// TIA Portal project "Lift_2026" (V15.1)

(* hardware
DEVICE "S71500/ET200MP station_1"  S7-1500 station
   slot 0: "Rail_0"  Rack  6ES7 590-1***0-0AA0
   slot 1: "PLC_1"  CPU 1513-1 PN  6ES7 513-1AL02-0AB0  V2.6
      slot 3: "CPU display_1"  6ES7591-1AA00-0AA0
DEVICE "HMI_1"  KTP900 Basic PN
   slot 0: "HMI_1"  KTP900 Basic PN  6AV2 123-2JB03-0AX0  15.1.0.0
   slot 1: "HMI_RT_1"  KTP900 Basic PN  6AV2 123-2JB03-0AX0  15.1.0.0
   slot 5: "HMI_1.IE_CP_1"  PROFINET Interface  15.0.1.0
      slot 1: "PROFINET Interface_1"  PROFINET Interface
         slot 1: "Port_1"  Port
*)

// ===== PLC "PLC_1"  CPU 1513-1 PN =====

VAR_GLOBAL   // PLC tag table "Default tag table"
   "Clock_Byte" AT %MB0 : Byte;
   "Clock_10Hz" AT %M0.0 : Bool;
   "Clock_5Hz" AT %M0.1 : Bool;
   "Clock_2.5Hz" AT %M0.2 : Bool;
   "Clock_2Hz" AT %M0.3 : Bool;
   "Clock_1.25Hz" AT %M0.4 : Bool;
   "Clock_1Hz" AT %M0.5 : Bool;
   "Clock_0.625Hz" AT %M0.6 : Bool;
   "Clock_0.5Hz" AT %M0.7 : Bool;
END_VAR

DATA_BLOCK "Alarme"   // DB1
{ S7_Optimized_Access := 'TRUE' }
VERSION : 0.1
   VAR
      alarme_gather : Word;
      alarme_vect : Array[0..15] of Bool;
   END_VAR
BEGIN
END_DATA_BLOCK

DATA_BLOCK "Avarii"   // DB2
{ S7_Optimized_Access := 'TRUE' }
VERSION : 0.1
   VAR
      esd : Bool;
      btn_esd : Bool;
      reset_esd : Bool;
      avarie_generala : Bool;
      reset_avarie_generala : Bool;
      avarie_usa : Bool;
      avarie_lumina : Bool;
      avarie_motor : Bool;
      avarie_greutate : Bool;
   END_VAR
BEGIN
END_DATA_BLOCK

DATA_BLOCK "Usa_Lift_DB"   // DB3
{ S7_Optimized_Access := 'TRUE' }
VERSION : 0.1
   VAR
      btn_urgenta : Bool;
      deschide_usa : Bool;
      inchide_usa : Bool;
      usa_deschisa : Bool;
      usa_inchisa : Bool;
   END_VAR
BEGIN
END_DATA_BLOCK

DATA_BLOCK "Bec_DB"   // DB4
{ S7_Optimized_Access := 'TRUE' }
VERSION : 0.1
   VAR
      permisiune_pornire : Bool;
      led_aprins : Bool;
   END_VAR
BEGIN
END_DATA_BLOCK

DATA_BLOCK "Motor_DB"   // DB5
{ S7_Optimized_Access := 'TRUE' }
VERSION : 0.1
   VAR
      pornire_stea : Bool;
      pornire_triunghi : Bool;
      directie_sus : Bool;
      directie_jos : Bool;
      permisiune_plecare : Bool;
   END_VAR
BEGIN
END_DATA_BLOCK

DATA_BLOCK "Simulare_DB"   // DB6
{ S7_Optimized_Access := 'TRUE' }
VERSION : 0.1
   VAR
      directie : USInt;
      etaj_curent : Int := 1;
      etaj_dorit : Int;
      etaj_chemat : Int;
      lift_in_miscare : Bool;
      btn_chemare_1 : Bool;
      btn_chemare_2 : Bool;
      btn_chemare_3 : Bool;
      btn_lift_1 : Bool;
      btn_lift_2 : Bool;
      btn_lift_3 : Bool;
      btn_add_pers : Bool;
      btn_sub_pers : Bool;
      time_elapsed_1 : Time;
      time_elapsed_2 : Time;
      time_elapsed_3 : Time;
      time_elapsed_4 : Time;
      time_elapsed_secunde_1 : Time;
      time_elapsed_secunde_2 : Time;
      time_elapsed_secunde_3 : Time;
      time_elapsed_secunde_4 : Time;
      "10s_cerut" : Bool;
      "10s_dorit" : Bool;
   END_VAR
BEGIN
END_DATA_BLOCK

DATA_BLOCK "Senzor_greutate_DB"   // DB7
{ S7_Optimized_Access := 'TRUE' }
VERSION : 0.1
   VAR
      permisiune_plecare : Bool := true;
      greutate_maxima : Real := 300.0;
      greutate_curenta : Real;
      greutate_depasita : Bool;
   END_VAR
BEGIN
END_DATA_BLOCK

DATA_BLOCK "Bec_DB_1"   // DB10
{ S7_Optimized_Access := 'TRUE' }
VERSION : 0.1
// stored: InstanceOfName Bec
"Bec"
BEGIN
END_DATA_BLOCK

DATA_BLOCK "Usa_Lift_DB_1"   // DB11
{ S7_Optimized_Access := 'TRUE' }
VERSION : 0.1
// stored: InstanceOfName Usa
"Usa"
BEGIN
END_DATA_BLOCK

DATA_BLOCK "Usa_Et_1_DB"   // DB12
{ S7_Optimized_Access := 'TRUE' }
VERSION : 0.1
   VAR
      deschide_usa : Bool;
      inchide_usa : Bool;
      usa_deschisa : Bool;
      usa_inchisa : Bool;
      btn_urgenta : Bool;
   END_VAR
BEGIN
END_DATA_BLOCK

DATA_BLOCK "USa_Et_2_DB"   // DB13
{ S7_Optimized_Access := 'TRUE' }
VERSION : 0.1
   VAR
      btn_urgenta : Bool;
      deschide_usa : Bool;
      inchide_usa : Bool;
      usa_deschisa : Bool;
      usa_inchisa : Bool;
   END_VAR
BEGIN
END_DATA_BLOCK

DATA_BLOCK "Usa_Et_3_DB"   // DB14
{ S7_Optimized_Access := 'TRUE' }
VERSION : 0.1
   VAR
      btn_urgenta : Bool;
      deschide_usa : Bool;
      inchide_usa : Bool;
      usa_deschisa : Bool;
      usa_inchisa : Bool;
   END_VAR
BEGIN
END_DATA_BLOCK

DATA_BLOCK "Usa_Et_1_DB_1"   // DB15
{ S7_Optimized_Access := 'TRUE' }
VERSION : 0.1
// stored: InstanceOfName Usa
"Usa"
BEGIN
END_DATA_BLOCK

DATA_BLOCK "Usa_Et_2_DB_1"   // DB16
{ S7_Optimized_Access := 'TRUE' }
VERSION : 0.1
// stored: InstanceOfName Usa
"Usa"
BEGIN
END_DATA_BLOCK

DATA_BLOCK "Usa_Et_3_DB_1"   // DB17
{ S7_Optimized_Access := 'TRUE' }
VERSION : 0.1
// stored: InstanceOfName Usa
"Usa"
BEGIN
END_DATA_BLOCK

DATA_BLOCK "Senzor_greutate_DB_1"   // DB18
{ S7_Optimized_Access := 'TRUE' }
VERSION : 0.1
// stored: InstanceOfName Senzor_greutate
"Senzor_greutate"
BEGIN
END_DATA_BLOCK

DATA_BLOCK "Motor_DB_1"   // DB19
{ S7_Optimized_Access := 'TRUE' }
VERSION : 0.1
// stored: InstanceOfName Motor
"Motor"
BEGIN
END_DATA_BLOCK

DATA_BLOCK "Simulare_DB_1"   // DB20
{ S7_Optimized_Access := 'TRUE' }
VERSION : 0.1
// stored: InstanceOfName Simulare
"Simulare"
BEGIN
END_DATA_BLOCK

// folder: System blocks/Program resources

DATA_BLOCK "timer_reset_esd"   // DB8
{ S7_Optimized_Access := 'TRUE' }
AUTHOR : Simatic
FAMILY : IEC
NAME : IEC_TMR
VERSION : 1.0
// stored: InstanceOfName IEC_TIMER
"IEC_TIMER"
BEGIN
END_DATA_BLOCK

DATA_BLOCK "timer_reset_avarie_generala"   // DB9
{ S7_Optimized_Access := 'TRUE' }
AUTHOR : Simatic
FAMILY : IEC
NAME : IEC_TMR
VERSION : 1.0
// stored: InstanceOfName IEC_TIMER
"IEC_TIMER"
BEGIN
END_DATA_BLOCK

// folder: (top level)

FUNCTION_BLOCK "Usa"   // FB1, LAD
{ S7_Optimized_Access := 'TRUE' }
VERSION : 0.1
   VAR_OUTPUT
      usa_deschisa : Bool;
      usa_inchisa : Bool;
   END_VAR
   VAR_IN_OUT
      deschide_usa : Bool;
      inchide_usa : Bool;
   END_VAR
   VAR
      timer_usa_inchisa : TON_TIME;
      timer_usa_deschisa : TON_TIME;
   END_VAR
BEGIN

REGION Network 1: deschide usa
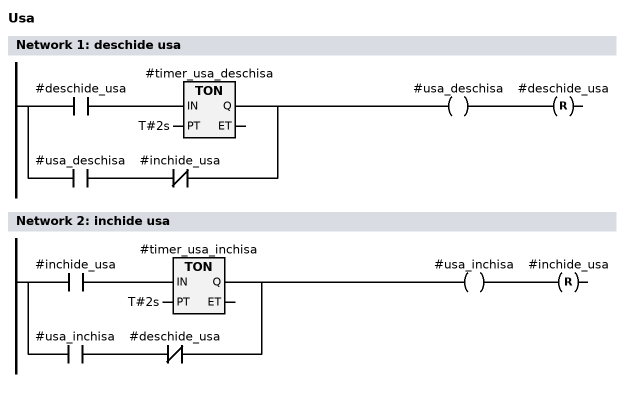
   #timer_usa_deschisa(IN := #deschide_usa, PT := T#2s);   // TON
   #usa_deschisa := #timer_usa_deschisa.Q OR (#usa_deschisa AND NOT #inchide_usa);
   IF #usa_deschisa THEN #deschide_usa := FALSE; END_IF;
END_REGION

REGION Network 2: inchide usa
   #timer_usa_inchisa(IN := #inchide_usa, PT := T#2s);   // TON
   #usa_inchisa := #timer_usa_inchisa.Q OR (#usa_inchisa AND NOT #deschide_usa);
   IF #usa_inchisa THEN #inchide_usa := FALSE; END_IF;
END_REGION
END_FUNCTION_BLOCK

FUNCTION_BLOCK "Bec"   // FB2, LAD
{ S7_Optimized_Access := 'TRUE' }
VERSION : 0.1
   VAR_INPUT
      permisiune_pornire : Bool;
   END_VAR
   VAR_OUTPUT
      bec_aprins : Bool;
   END_VAR
BEGIN

REGION Network 1
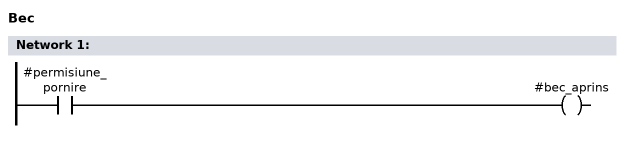
   RUNG wire#powerrail
      Contact( #permisiune_pornire )
      Coil( #bec_aprins )
   END_RUNG
   // the same network as SCL:
   #bec_aprins := #permisiune_pornire;
END_REGION
END_FUNCTION_BLOCK

FUNCTION_BLOCK "Motor"   // FB3, LAD
{ S7_Optimized_Access := 'TRUE' }
VERSION : 0.1
   VAR_INPUT
      directie : USInt;
   END_VAR
   VAR_OUTPUT
      pornire_stea : Bool;
      pornire_triunghi : Bool;
      directie_sus : Bool;
      directie_jos : Bool;
   END_VAR
   VAR_IN_OUT
      permisiune_plecare : Bool;
   END_VAR
   VAR
      timer_stea : TON_TIME;
   END_VAR
BEGIN

REGION Network 1: Selecteaza directia
   // simulata cu valori algebrice, insa in mod normal ar fi un contact pentru directie, depinzand cum se conecteaza, selecteaza directia, insa pentru simplitate am optat la asta
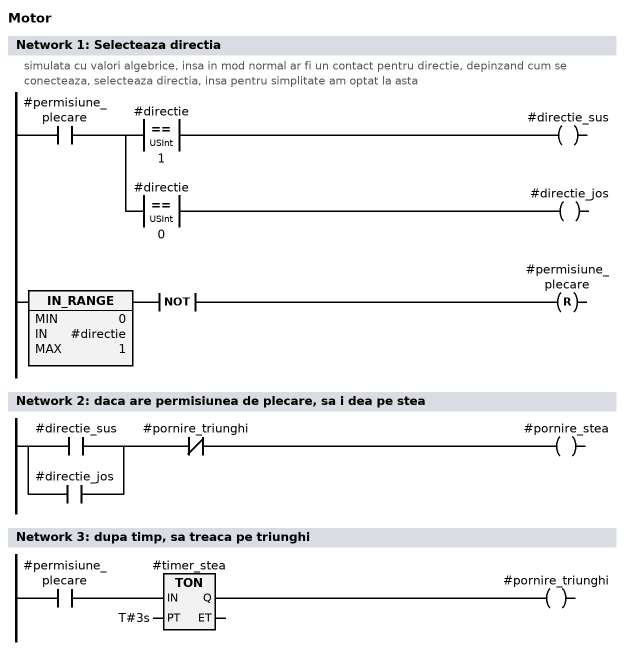
   RUNG wire#powerrail
      Contact( #permisiune_plecare )
      wire#w1
      { S7_Templates := "SrcType := USInt" } EQ_Contact(in1 := #directie, in2 := 1)
      Coil( #directie_sus )
   END_RUNG
   RUNG wire#w1
      { S7_Templates := "SrcType := USInt" } EQ_Contact(in1 := #directie, in2 := 0)
      Coil( #directie_jos )
   END_RUNG
   RUNG wire#powerrail
      { S7_Templates := "SrcType := USInt" } InRange(min := 0, in := #directie, max := 1)
      Not()
      R_Coil( #permisiune_plecare )
   END_RUNG
   // the same network as SCL:
   #directie_sus := #permisiune_plecare AND (#directie = 1);
   #directie_jos := #permisiune_plecare AND (#directie = 0);
   IF NOT ((0 <= #directie) AND (#directie <= 1)) THEN #permisiune_plecare := FALSE; END_IF;
END_REGION

REGION Network 2: daca are permisiunea de plecare, sa i dea pe stea
   RUNG wire#powerrail
      Contact( #directie_sus )
      wire#w1
      I_Contact( #pornire_triunghi )
      Coil( #pornire_stea )
   END_RUNG
   RUNG wire#powerrail
      Contact( #directie_jos )
   END_RUNG wire#w1
   // the same network as SCL:
   #pornire_stea := (#directie_sus OR #directie_jos) AND NOT #pornire_triunghi;
END_REGION

REGION Network 3: dupa timp, sa treaca pe triunghi
   #timer_stea(IN := #permisiune_plecare, PT := T#3s);   // TON
   #pornire_triunghi := #timer_stea.Q;
END_REGION
END_FUNCTION_BLOCK

FUNCTION_BLOCK "Simulare"   // FB4, LAD
{ S7_Optimized_Access := 'TRUE' }
VERSION : 0.1
   VAR_INPUT
      motor_pornit : Bool;
      greutate_maxima : Real;
      greutate_depasita : Bool;
      esd : Bool;
      avarie_generala : Bool;
      este_deschis_1 : Bool;
      este_deschis_2 : Bool;
      este_deschis_3 : Bool;
   END_VAR
   VAR_OUTPUT
      directie : USInt;
      lift_in_miscare : Bool;
      time_elapsed_dorit_1 : Time;
      time_elapsed_dorit_2 : Time;
      time_elapsed_cerut_1 : Time;
      time_elapsed_cerut_2 : Time;
      "10s_dorit" : Bool;
      "10s_cerut" : Bool;
   END_VAR
   VAR_IN_OUT
      btn_urgenta_usa_1 : Bool;
      btn_urgenta_usa_2 : Bool;
      btn_urgenta_usa_3 : Bool;
      btn_urgenta_usa_lift : Bool;
      btn_add_pers : Bool;
      btn_sub_pers : Bool;
      usa_lift_inchisa : Bool;
      usa_lift_deschisa : Bool;
      usa_deschisa_et_1 : Bool;
      usa_deschisa_et_2 : Bool;
      usa_deschisa_et_3 : Bool;
      usa_inchisa_et_1 : Bool;
      usa_inchisa_et_2 : Bool;
      usa_inchisa_et_3 : Bool;
      plecare_motor : Bool;
      plecare_greutate : Bool;
      plecare_lumina : Bool;
      btn_chemare_1 : Bool;
      btn_chemare_2 : Bool;
      btn_chemare_3 : Bool;
      btn_lift_1 : Bool;
      btn_lift_2 : Bool;
      btn_lift_3 : Bool;
      etaj_curent : Int;
      etaj_dorit : Int;
      etaj_chemat : Int;
      greutate_curenta : Real;
   END_VAR
   VAR
      ajuns_chemare : Bool;
      plecare : Bool;
      terminat_proces : Bool;
      timer_5s_chemat : TON_TIME;
      timer_10s_chemat : TON_TIME;
      timer_5s_plecat : TON_TIME;
      timer_10s_plecat : TON_TIME;
      timer_resetare_terminare : TON_TIME;
      add : Bool;
      sub : Bool;
      diferenta_chemat : Int;
      diferenta_plecat : Int;
      re_add : Bool;
      re_sub : Bool;
      trm_5s_plecat : Bool;
      trm_10s_plecat : Bool;
      trm_plecat : Bool;
      trm_5s_chemat : Bool;
      trm_10s_chemat : Bool;
      trm_chemat : Bool;
   END_VAR
   VAR_TEMP   // added for the SCL form of the ladder/FBD networks
      _w1 : Bool;
      _w2 : Bool;
      _w3 : Bool;
   END_VAR
BEGIN

REGION Network 1: seteaza ca liftul e in miscare
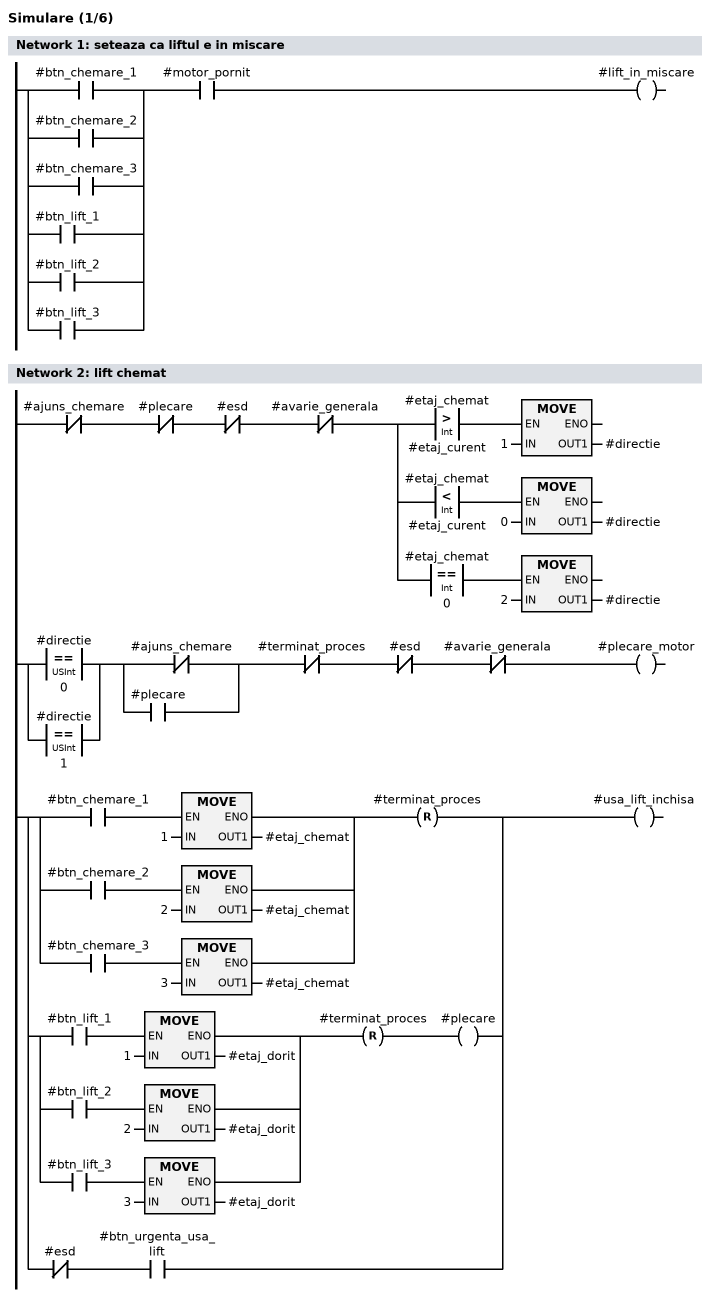
   RUNG wire#powerrail
      Contact( #btn_chemare_1 )
      wire#w1
      Contact( #motor_pornit )
      Coil( #lift_in_miscare )
   END_RUNG
   RUNG wire#powerrail
      Contact( #btn_chemare_2 )
   END_RUNG wire#w1
   RUNG wire#powerrail
      Contact( #btn_chemare_3 )
   END_RUNG wire#w1
   RUNG wire#powerrail
      Contact( #btn_lift_1 )
   END_RUNG wire#w1
   RUNG wire#powerrail
      Contact( #btn_lift_2 )
   END_RUNG wire#w1
   RUNG wire#powerrail
      Contact( #btn_lift_3 )
   END_RUNG wire#w1
   // the same network as SCL:
   #lift_in_miscare := (#btn_chemare_1 OR #btn_chemare_2 OR #btn_chemare_3 OR #btn_lift_1 OR #btn_lift_2 OR #btn_lift_3) AND #motor_pornit;
END_REGION

REGION Network 2: lift chemat
   RUNG wire#powerrail
      I_Contact( #ajuns_chemare )
      I_Contact( #plecare )
      I_Contact( #esd )
      I_Contact( #avarie_generala )
      wire#w1
      { S7_Templates := "SrcType := Int" } GT_Contact(in1 := #etaj_chemat, in2 := #etaj_curent)
      Move(in := 1, out1 => #directie)
   END_RUNG
   RUNG wire#w1
      { S7_Templates := "SrcType := Int" } LT_Contact(in1 := #etaj_chemat, in2 := #etaj_curent)
      Move(in := 0, out1 => #directie)
   END_RUNG
   RUNG wire#w1
      { S7_Templates := "SrcType := Int" } EQ_Contact(in1 := #etaj_chemat, in2 := 0)
      Move(in := 2, out1 => #directie)
   END_RUNG
   RUNG wire#powerrail
      { S7_Templates := "SrcType := USInt" } EQ_Contact(in1 := #directie, in2 := 0)
      wire#w2
      I_Contact( #ajuns_chemare )
      wire#w3
      I_Contact( #terminat_proces )
      I_Contact( #esd )
      I_Contact( #avarie_generala )
      Coil( #plecare_motor )
   END_RUNG
   RUNG wire#powerrail
      { S7_Templates := "SrcType := USInt" } EQ_Contact(in1 := #directie, in2 := 1)
   END_RUNG wire#w2
   RUNG wire#w2
      Contact( #plecare )
   END_RUNG wire#w3
   RUNG wire#powerrail
      Contact( #btn_chemare_1 )
      Move(in := 1, out1 => #etaj_chemat)
      wire#w4
      R_Coil( #terminat_proces )
      wire#w5
      Coil( #usa_lift_inchisa )
   END_RUNG
   RUNG wire#powerrail
      Contact( #btn_chemare_2 )
      Move(in := 2, out1 => #etaj_chemat)
   END_RUNG wire#w4
   RUNG wire#powerrail
      Contact( #btn_chemare_3 )
      Move(in := 3, out1 => #etaj_chemat)
   END_RUNG wire#w4
   RUNG wire#powerrail
      Contact( #btn_lift_1 )
      Move(in := 1, out1 => #etaj_dorit)
      wire#w6
      R_Coil( #terminat_proces )
      Coil( #plecare )
   END_RUNG wire#w5
   RUNG wire#powerrail
      Contact( #btn_lift_2 )
      Move(in := 2, out1 => #etaj_dorit)
   END_RUNG wire#w6
   RUNG wire#powerrail
      Contact( #btn_lift_3 )
      Move(in := 3, out1 => #etaj_dorit)
   END_RUNG wire#w6
   RUNG wire#powerrail
      I_Contact( #esd )
      Contact( #btn_urgenta_usa_lift )
   END_RUNG wire#w5
   // the same network as SCL:
   #_w1 := NOT #ajuns_chemare AND NOT #plecare AND NOT #esd AND NOT #avarie_generala;
   IF #_w1 AND (#etaj_chemat > #etaj_curent) THEN #directie := 1; END_IF;
   IF #_w1 AND (#etaj_chemat < #etaj_curent) THEN #directie := 0; END_IF;
   IF #_w1 AND (#etaj_chemat = 0) THEN #directie := 2; END_IF;
   #plecare_motor := ((#directie = 0) OR (#directie = 1)) AND (NOT #ajuns_chemare OR #plecare) AND NOT #terminat_proces AND NOT #esd AND NOT #avarie_generala;
   IF #btn_chemare_1 THEN #etaj_chemat := 1; END_IF;
   IF #btn_chemare_2 THEN #etaj_chemat := 2; END_IF;
   IF #btn_chemare_3 THEN #etaj_chemat := 3; END_IF;
   #_w2 := #btn_chemare_1 OR #btn_chemare_2 OR #btn_chemare_3;
   IF #_w2 THEN #terminat_proces := FALSE; END_IF;
   IF #btn_lift_1 THEN #etaj_dorit := 1; END_IF;
   IF #btn_lift_2 THEN #etaj_dorit := 2; END_IF;
   IF #btn_lift_3 THEN #etaj_dorit := 3; END_IF;
   #_w3 := #btn_lift_1 OR #btn_lift_2 OR #btn_lift_3;
   IF #_w3 THEN #terminat_proces := FALSE; END_IF;
   #plecare := #_w3;
   #usa_lift_inchisa := #_w2 OR #_w3 OR (NOT #esd AND #btn_urgenta_usa_lift);
END_REGION

REGION Network 3: daca simte persoana, aprinde lumina (pentru simplitate :) ), si calculeaza si diferenta, cuz why not
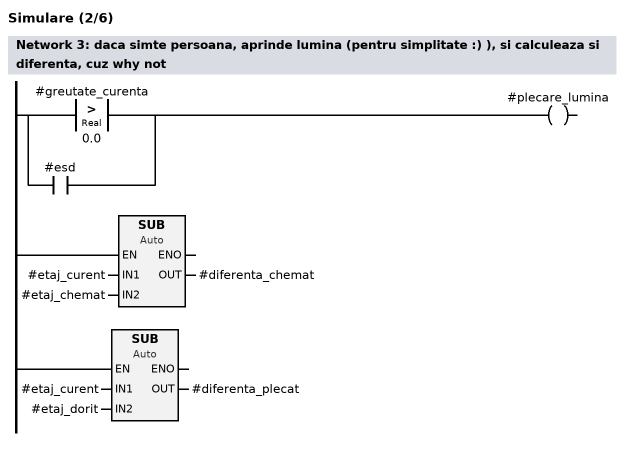
   RUNG wire#powerrail
      { S7_Templates := "SrcType := Real" } GT_Contact(in1 := #greutate_curenta, in2 := 0.0)
      wire#w1
      Coil( #plecare_lumina )
   END_RUNG
   RUNG wire#powerrail
      Contact( #esd )
   END_RUNG wire#w1
   RUNG wire#powerrail
      Sub(in1 := #etaj_curent, in2 := #etaj_chemat, out => #diferenta_chemat)
   END_RUNG
   RUNG wire#powerrail
      Sub(in1 := #etaj_curent, in2 := #etaj_dorit, out => #diferenta_plecat)
   END_RUNG
   // the same network as SCL:
   #plecare_lumina := (#greutate_curenta > 0.0) OR #esd;
   #diferenta_chemat := #etaj_curent - #etaj_chemat;
   #diferenta_plecat := #etaj_curent - #etaj_dorit;
END_REGION

REGION Network 4: daca a pornit motorul, depinzand de diferenta, pune ton ul
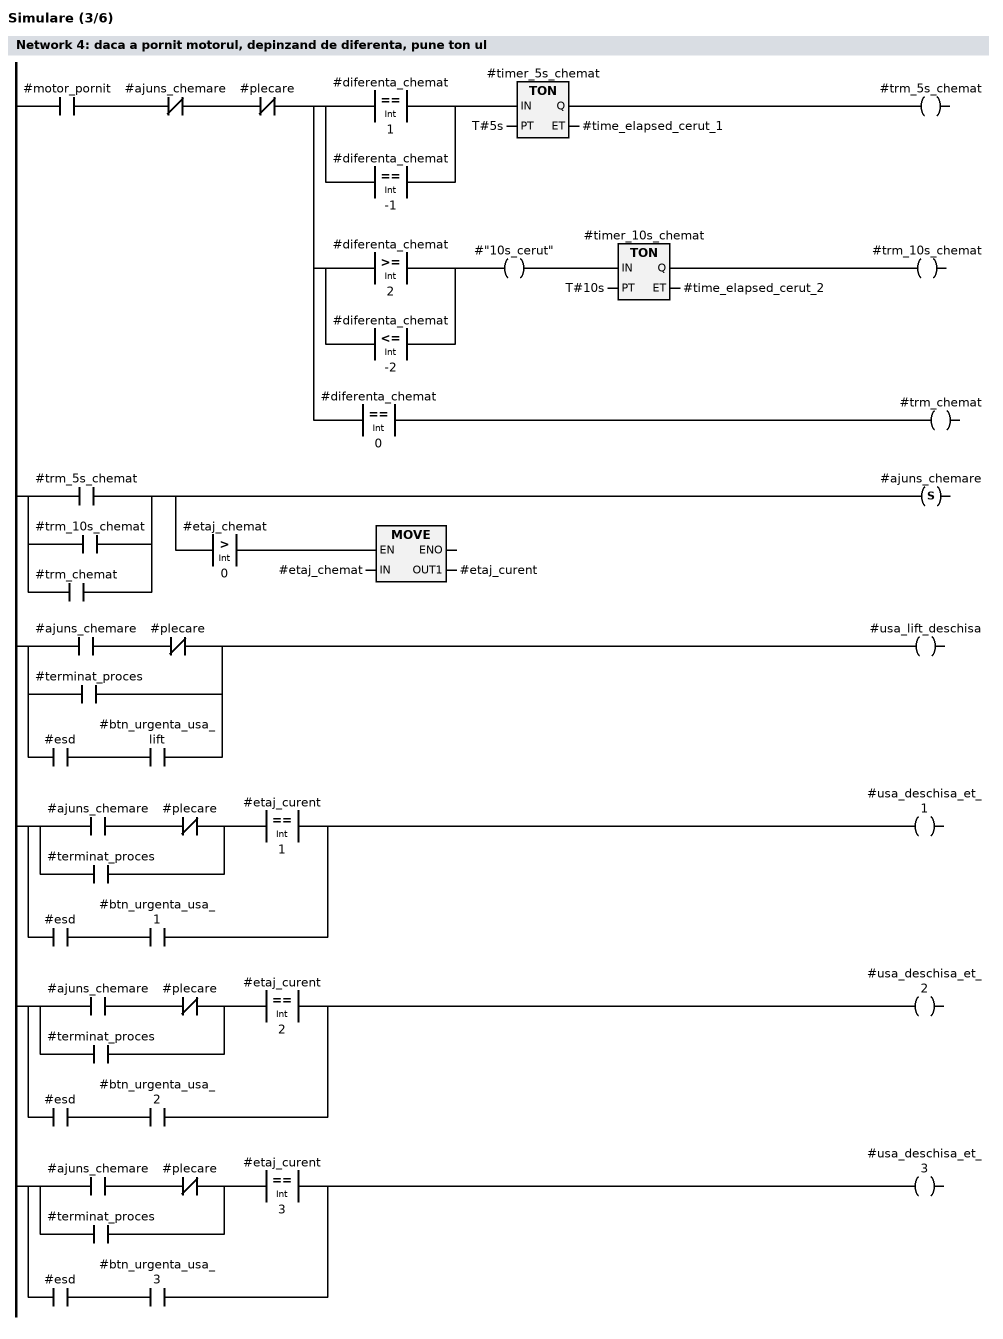
   #_w1 := #motor_pornit AND NOT #ajuns_chemare AND NOT #plecare;
   #timer_5s_chemat(IN := #_w1 AND ((#diferenta_chemat = 1) OR (#diferenta_chemat = (-1))),   // TON
                    PT := T#5s,
                    ET => #time_elapsed_cerut_1);
   #trm_5s_chemat := #timer_5s_chemat.Q;
   #"10s_cerut" := #_w1 AND ((#diferenta_chemat >= 2) OR (#diferenta_chemat <= (-2)));
   #timer_10s_chemat(IN := #"10s_cerut", PT := T#10s, ET => #time_elapsed_cerut_2);   // TON
   #trm_10s_chemat := #timer_10s_chemat.Q;
   #trm_chemat := #_w1 AND (#diferenta_chemat = 0);
   #_w2 := #trm_5s_chemat OR #trm_10s_chemat OR #trm_chemat;
   IF #_w2 THEN #ajuns_chemare := TRUE; END_IF;
   IF #_w2 AND (#etaj_chemat > 0) THEN #etaj_curent := #etaj_chemat; END_IF;
   #usa_lift_deschisa := (#ajuns_chemare AND NOT #plecare) OR #terminat_proces OR (#esd AND #btn_urgenta_usa_lift);
   #usa_deschisa_et_1 := (((#ajuns_chemare AND NOT #plecare) OR #terminat_proces) AND (#etaj_curent = 1)) OR (#esd AND #btn_urgenta_usa_1);
   #usa_deschisa_et_2 := (((#ajuns_chemare AND NOT #plecare) OR #terminat_proces) AND (#etaj_curent = 2)) OR (#esd AND #btn_urgenta_usa_2);
   #usa_deschisa_et_3 := (((#ajuns_chemare AND NOT #plecare) OR #terminat_proces) AND (#etaj_curent = 3)) OR (#esd AND #btn_urgenta_usa_3);
END_REGION

REGION Network 5: daca ii da buton din lift, sa plece la fel
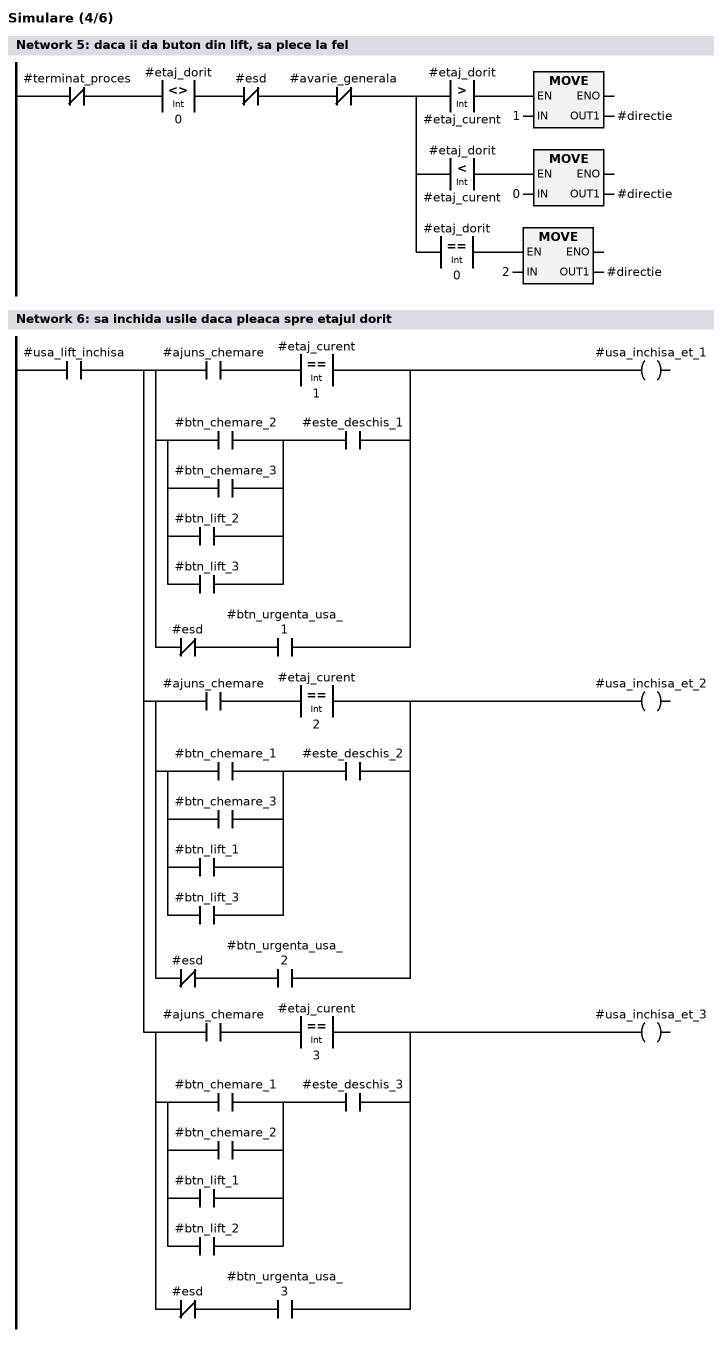
   RUNG wire#powerrail
      I_Contact( #terminat_proces )
      { S7_Templates := "SrcType := Int" } NE_Contact(in1 := #etaj_dorit, in2 := 0)
      I_Contact( #esd )
      I_Contact( #avarie_generala )
      wire#w1
      { S7_Templates := "SrcType := Int" } GT_Contact(in1 := #etaj_dorit, in2 := #etaj_curent)
      Move(in := 1, out1 => #directie)
   END_RUNG
   RUNG wire#w1
      { S7_Templates := "SrcType := Int" } LT_Contact(in1 := #etaj_dorit, in2 := #etaj_curent)
      Move(in := 0, out1 => #directie)
   END_RUNG
   RUNG wire#w1
      { S7_Templates := "SrcType := Int" } EQ_Contact(in1 := #etaj_dorit, in2 := 0)
      Move(in := 2, out1 => #directie)
   END_RUNG
   // the same network as SCL:
   #_w1 := NOT #terminat_proces AND (#etaj_dorit <> 0) AND NOT #esd AND NOT #avarie_generala;
   IF #_w1 AND (#etaj_dorit > #etaj_curent) THEN #directie := 1; END_IF;
   IF #_w1 AND (#etaj_dorit < #etaj_curent) THEN #directie := 0; END_IF;
   IF #_w1 AND (#etaj_dorit = 0) THEN #directie := 2; END_IF;
END_REGION

REGION Network 6: sa inchida usile daca pleaca spre etajul dorit
   RUNG wire#powerrail
      Contact( #usa_lift_inchisa )
      wire#w1
      Contact( #ajuns_chemare )
      { S7_Templates := "SrcType := Int" } EQ_Contact(in1 := #etaj_curent, in2 := 1)
      wire#w2
      Coil( #usa_inchisa_et_1 )
   END_RUNG
   RUNG wire#w1
      Contact( #btn_chemare_2 )
      wire#w3
      Contact( #este_deschis_1 )
   END_RUNG wire#w2
   RUNG wire#w1
      Contact( #btn_chemare_3 )
   END_RUNG wire#w3
   RUNG wire#w1
      Contact( #btn_lift_2 )
   END_RUNG wire#w3
   RUNG wire#w1
      Contact( #btn_lift_3 )
   END_RUNG wire#w3
   RUNG wire#w1
      I_Contact( #esd )
      Contact( #btn_urgenta_usa_1 )
   END_RUNG wire#w2
   RUNG wire#w1
      Contact( #ajuns_chemare )
      { S7_Templates := "SrcType := Int" } EQ_Contact(in1 := #etaj_curent, in2 := 2)
      wire#w4
      Coil( #usa_inchisa_et_2 )
   END_RUNG
   RUNG wire#w1
      Contact( #btn_chemare_1 )
      wire#w5
      Contact( #este_deschis_2 )
   END_RUNG wire#w4
   RUNG wire#w1
      Contact( #btn_chemare_3 )
   END_RUNG wire#w5
   RUNG wire#w1
      Contact( #btn_lift_1 )
   END_RUNG wire#w5
   RUNG wire#w1
      Contact( #btn_lift_3 )
   END_RUNG wire#w5
   RUNG wire#w1
      I_Contact( #esd )
      Contact( #btn_urgenta_usa_2 )
   END_RUNG wire#w4
   RUNG wire#w1
      Contact( #ajuns_chemare )
      { S7_Templates := "SrcType := Int" } EQ_Contact(in1 := #etaj_curent, in2 := 3)
      wire#w6
      Coil( #usa_inchisa_et_3 )
   END_RUNG
   RUNG wire#w1
      Contact( #btn_chemare_1 )
      wire#w7
      Contact( #este_deschis_3 )
   END_RUNG wire#w6
   RUNG wire#w1
      Contact( #btn_chemare_2 )
   END_RUNG wire#w7
   RUNG wire#w1
      Contact( #btn_lift_1 )
   END_RUNG wire#w7
   RUNG wire#w1
      Contact( #btn_lift_2 )
   END_RUNG wire#w7
   RUNG wire#w1
      I_Contact( #esd )
      Contact( #btn_urgenta_usa_3 )
   END_RUNG wire#w6
   // the same network as SCL:
   #usa_inchisa_et_1 := #usa_lift_inchisa AND ((#ajuns_chemare AND (#etaj_curent = 1)) OR ((#btn_chemare_2 OR #btn_chemare_3 OR #btn_lift_2 OR #btn_lift_3) AND #este_deschis_1) OR (NOT #esd AND #btn_urgenta_usa_1));
   #usa_inchisa_et_2 := #usa_lift_inchisa AND ((#ajuns_chemare AND (#etaj_curent = 2)) OR ((#btn_chemare_1 OR #btn_chemare_3 OR #btn_lift_1 OR #btn_lift_3) AND #este_deschis_2) OR (NOT #esd AND #btn_urgenta_usa_2));
   #usa_inchisa_et_3 := #usa_lift_inchisa AND ((#ajuns_chemare AND (#etaj_curent = 3)) OR ((#btn_chemare_1 OR #btn_chemare_2 OR #btn_lift_1 OR #btn_lift_2) AND #este_deschis_3) OR (NOT #esd AND #btn_urgenta_usa_3));
END_REGION

REGION Network 7: daca a pornit motorul, sa mearga la etajul dorit
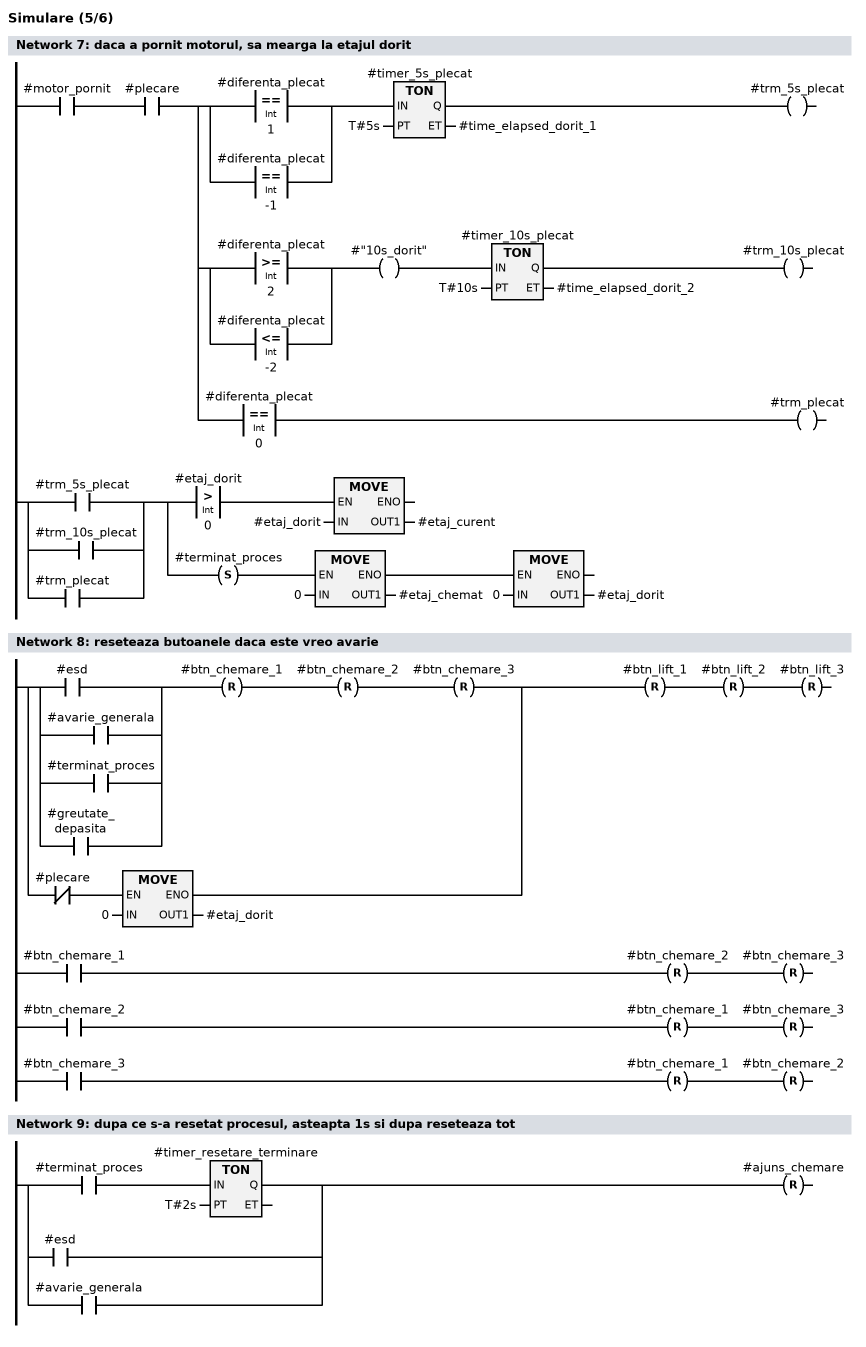
   #_w1 := #motor_pornit AND #plecare;
   #timer_5s_plecat(IN := #_w1 AND ((#diferenta_plecat = 1) OR (#diferenta_plecat = (-1))),   // TON
                    PT := T#5s,
                    ET => #time_elapsed_dorit_1);
   #trm_5s_plecat := #timer_5s_plecat.Q;
   #"10s_dorit" := #_w1 AND ((#diferenta_plecat >= 2) OR (#diferenta_plecat <= (-2)));
   #timer_10s_plecat(IN := #"10s_dorit", PT := T#10s, ET => #time_elapsed_dorit_2);   // TON
   #trm_10s_plecat := #timer_10s_plecat.Q;
   #trm_plecat := #_w1 AND (#diferenta_plecat = 0);
   #_w2 := #trm_5s_plecat OR #trm_10s_plecat OR #trm_plecat;
   IF #_w2 AND (#etaj_dorit > 0) THEN #etaj_curent := #etaj_dorit; END_IF;
   IF #_w2 THEN
       #terminat_proces := TRUE;
       #etaj_chemat := 0;
       #etaj_dorit := 0;
   END_IF;
END_REGION

REGION Network 8: reseteaza butoanele daca este vreo avarie
   RUNG wire#powerrail
      Contact( #esd )
      wire#w1
      R_Coil( #btn_chemare_1 )
      R_Coil( #btn_chemare_2 )
      R_Coil( #btn_chemare_3 )
      wire#w2
      R_Coil( #btn_lift_1 )
      R_Coil( #btn_lift_2 )
      R_Coil( #btn_lift_3 )
   END_RUNG
   RUNG wire#powerrail
      Contact( #avarie_generala )
   END_RUNG wire#w1
   RUNG wire#powerrail
      Contact( #terminat_proces )
   END_RUNG wire#w1
   RUNG wire#powerrail
      Contact( #greutate_depasita )
   END_RUNG wire#w1
   RUNG wire#powerrail
      I_Contact( #plecare )
      Move(in := 0, out1 => #etaj_dorit)
   END_RUNG wire#w2
   RUNG wire#powerrail
      Contact( #btn_chemare_1 )
      R_Coil( #btn_chemare_2 )
      R_Coil( #btn_chemare_3 )
   END_RUNG
   RUNG wire#powerrail
      Contact( #btn_chemare_2 )
      R_Coil( #btn_chemare_1 )
      R_Coil( #btn_chemare_3 )
   END_RUNG
   RUNG wire#powerrail
      Contact( #btn_chemare_3 )
      R_Coil( #btn_chemare_1 )
      R_Coil( #btn_chemare_2 )
   END_RUNG
   // the same network as SCL:
   #_w1 := #esd OR #avarie_generala OR #terminat_proces OR #greutate_depasita;
   IF #_w1 THEN
       #btn_chemare_1 := FALSE;
       #btn_chemare_2 := FALSE;
       #btn_chemare_3 := FALSE;
   END_IF;
   IF NOT #plecare THEN #etaj_dorit := 0; END_IF;
   IF #_w1 OR NOT #plecare THEN
       #btn_lift_1 := FALSE;
       #btn_lift_2 := FALSE;
       #btn_lift_3 := FALSE;
   END_IF;
   IF #btn_chemare_1 THEN
       #btn_chemare_2 := FALSE;
       #btn_chemare_3 := FALSE;
   END_IF;
   IF #btn_chemare_2 THEN
       #btn_chemare_1 := FALSE;
       #btn_chemare_3 := FALSE;
   END_IF;
   IF #btn_chemare_3 THEN
       #btn_chemare_1 := FALSE;
       #btn_chemare_2 := FALSE;
   END_IF;
END_REGION

REGION Network 9: dupa ce s-a resetat procesul, asteapta 1s si dupa reseteaza tot
   #timer_resetare_terminare(IN := #terminat_proces, PT := T#2s);   // TON
   IF #timer_resetare_terminare.Q OR #esd OR #avarie_generala THEN #ajuns_chemare := FALSE; END_IF;
END_REGION

REGION Network 10: butoane pt a adauga/scoate persoane din lift
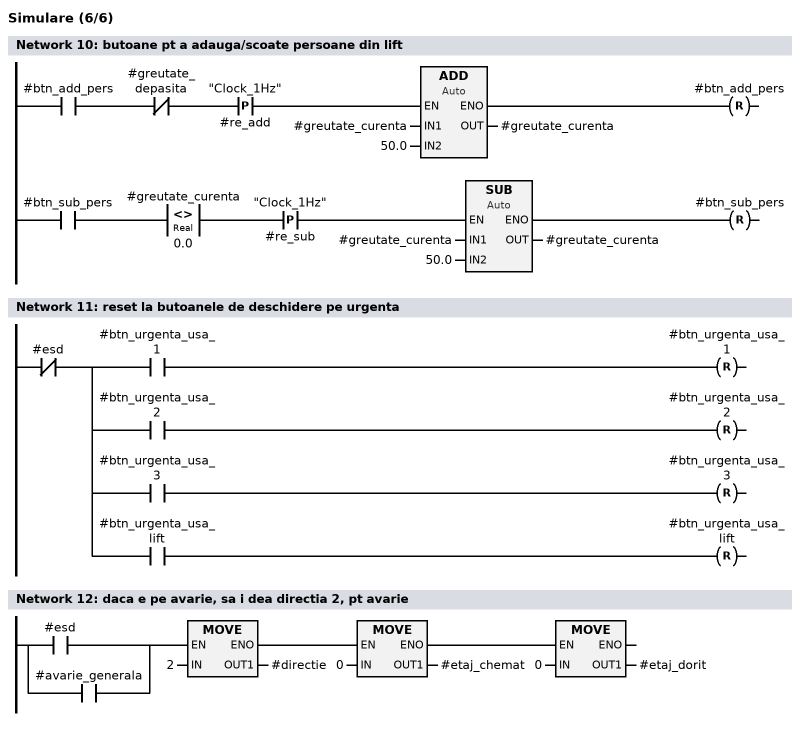
   RUNG wire#powerrail
      Contact( #btn_add_pers )
      I_Contact( #greutate_depasita )
      P_Contact(operand := "Clock_1Hz", bit := #re_add)
      Add(in1 := #greutate_curenta, in2 := 50.0, out => #greutate_curenta)
      R_Coil( #btn_add_pers )
   END_RUNG
   RUNG wire#powerrail
      Contact( #btn_sub_pers )
      { S7_Templates := "SrcType := Real" } NE_Contact(in1 := #greutate_curenta, in2 := 0.0)
      P_Contact(operand := "Clock_1Hz", bit := #re_sub)
      Sub(in1 := #greutate_curenta, in2 := 50.0, out => #greutate_curenta)
      R_Coil( #btn_sub_pers )
   END_RUNG
   // the same network as SCL:
   #_w1 := #btn_add_pers AND NOT #greutate_depasita AND "Clock_1Hz" AND NOT #re_add;   // rising edge of "Clock_1Hz"
   #re_add := "Clock_1Hz";
   IF #_w1 THEN
       #greutate_curenta := #greutate_curenta + 50.0;
       #btn_add_pers := FALSE;
   END_IF;
   #_w2 := #btn_sub_pers AND (#greutate_curenta <> 0.0) AND "Clock_1Hz" AND NOT #re_sub;   // rising edge of "Clock_1Hz"
   #re_sub := "Clock_1Hz";
   IF #_w2 THEN
       #greutate_curenta := #greutate_curenta - 50.0;
       #btn_sub_pers := FALSE;
   END_IF;
END_REGION

REGION Network 11: reset la butoanele de deschidere pe urgenta
   RUNG wire#powerrail
      I_Contact( #esd )
      wire#w1
      Contact( #btn_urgenta_usa_1 )
      R_Coil( #btn_urgenta_usa_1 )
   END_RUNG
   RUNG wire#w1
      Contact( #btn_urgenta_usa_2 )
      R_Coil( #btn_urgenta_usa_2 )
   END_RUNG
   RUNG wire#w1
      Contact( #btn_urgenta_usa_3 )
      R_Coil( #btn_urgenta_usa_3 )
   END_RUNG
   RUNG wire#w1
      Contact( #btn_urgenta_usa_lift )
      R_Coil( #btn_urgenta_usa_lift )
   END_RUNG
   // the same network as SCL:
   IF NOT #esd AND #btn_urgenta_usa_1 THEN #btn_urgenta_usa_1 := FALSE; END_IF;
   IF NOT #esd AND #btn_urgenta_usa_2 THEN #btn_urgenta_usa_2 := FALSE; END_IF;
   IF NOT #esd AND #btn_urgenta_usa_3 THEN #btn_urgenta_usa_3 := FALSE; END_IF;
   IF NOT #esd AND #btn_urgenta_usa_lift THEN #btn_urgenta_usa_lift := FALSE; END_IF;
END_REGION

REGION Network 12: daca e pe avarie, sa i dea directia 2, pt avarie
   RUNG wire#powerrail
      Contact( #esd )
      wire#w1
      Move(in := 2, out1 => #directie)
      Move(in := 0, out1 => #etaj_chemat)
      Move(in := 0, out1 => #etaj_dorit)
   END_RUNG
   RUNG wire#powerrail
      Contact( #avarie_generala )
   END_RUNG wire#w1
   // the same network as SCL:
   IF #esd OR #avarie_generala THEN
       #directie := 2;
       #etaj_chemat := 0;
       #etaj_dorit := 0;
   END_IF;
END_REGION
END_FUNCTION_BLOCK

FUNCTION_BLOCK "Senzor_greutate"   // FB5, LAD
{ S7_Optimized_Access := 'TRUE' }
VERSION : 0.1
   VAR_INPUT
      permisiune_plecare : Bool;
      greutate_maxima : Real;
   END_VAR
   VAR_OUTPUT
      greutate_depasita : Bool;
   END_VAR
   VAR_IN_OUT
      greutate_curenta : Real;
   END_VAR
   VAR
      pornit : Bool;
   END_VAR
BEGIN

REGION Network 1: daca are permisiune de plecare,
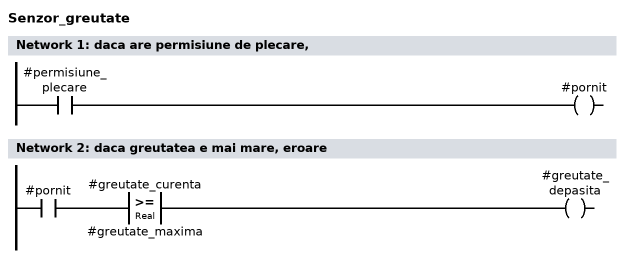
   RUNG wire#powerrail
      Contact( #permisiune_plecare )
      Coil( #pornit )
   END_RUNG
   // the same network as SCL:
   #pornit := #permisiune_plecare;
END_REGION

REGION Network 2: daca greutatea e mai mare, eroare
   RUNG wire#powerrail
      Contact( #pornit )
      { S7_Templates := "SrcType := Real" } GE_Contact(in1 := #greutate_curenta, in2 := #greutate_maxima)
      Coil( #greutate_depasita )
   END_RUNG
   // the same network as SCL:
   #greutate_depasita := #pornit AND (#greutate_curenta >= #greutate_maxima);
END_REGION
END_FUNCTION_BLOCK

ORGANIZATION_BLOCK "Main"   // OB1, LAD, ProgramCycle
TITLE = "Main Program Sweep (Cycle)"
{ S7_Optimized_Access := 'TRUE' }
VERSION : 0.1
   VAR_INPUT
      Initial_Call : Bool;   // Initial call of this OB
      Remanence : Bool;   // =True, if remanent data are available
   END_VAR
BEGIN

REGION Network 1: Alarme gather
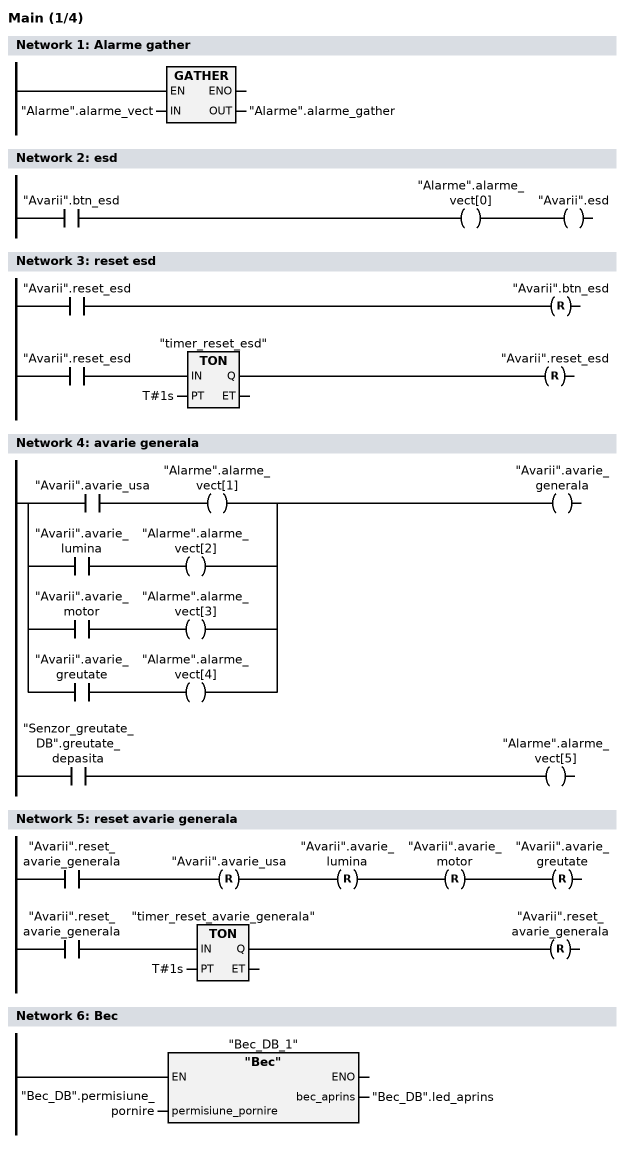
   GATHER(IN := "Alarme".alarme_vect, OUT => "Alarme".alarme_gather);
END_REGION

REGION Network 2: esd
   RUNG wire#powerrail
      Contact( "Avarii".btn_esd )
      Coil( "Alarme".alarme_vect[0] )
      Coil( "Avarii".esd )
   END_RUNG
   // the same network as SCL:
   "Alarme".alarme_vect[0] := "Avarii".btn_esd;
   "Avarii".esd := "Avarii".btn_esd;
END_REGION

REGION Network 3: reset esd
   IF "Avarii".reset_esd THEN "Avarii".btn_esd := FALSE; END_IF;
   "timer_reset_esd".TON(IN := "Avarii".reset_esd, PT := T#1s);
   IF "timer_reset_esd".Q THEN "Avarii".reset_esd := FALSE; END_IF;
END_REGION

REGION Network 4: avarie generala
   RUNG wire#powerrail
      Contact( "Avarii".avarie_usa )
      Coil( "Alarme".alarme_vect[1] )
      wire#w1
      Coil( "Avarii".avarie_generala )
   END_RUNG
   RUNG wire#powerrail
      Contact( "Avarii".avarie_lumina )
      Coil( "Alarme".alarme_vect[2] )
   END_RUNG wire#w1
   RUNG wire#powerrail
      Contact( "Avarii".avarie_motor )
      Coil( "Alarme".alarme_vect[3] )
   END_RUNG wire#w1
   RUNG wire#powerrail
      Contact( "Avarii".avarie_greutate )
      Coil( "Alarme".alarme_vect[4] )
   END_RUNG wire#w1
   RUNG wire#powerrail
      Contact( "Senzor_greutate_DB".greutate_depasita )
      Coil( "Alarme".alarme_vect[5] )
   END_RUNG
   // the same network as SCL:
   "Alarme".alarme_vect[1] := "Avarii".avarie_usa;
   "Alarme".alarme_vect[2] := "Avarii".avarie_lumina;
   "Alarme".alarme_vect[3] := "Avarii".avarie_motor;
   "Alarme".alarme_vect[4] := "Avarii".avarie_greutate;
   "Avarii".avarie_generala := "Avarii".avarie_usa OR "Avarii".avarie_lumina OR "Avarii".avarie_motor OR "Avarii".avarie_greutate;
   "Alarme".alarme_vect[5] := "Senzor_greutate_DB".greutate_depasita;
END_REGION

REGION Network 5: reset avarie generala
   IF "Avarii".reset_avarie_generala THEN
       "Avarii".avarie_usa := FALSE;
       "Avarii".avarie_lumina := FALSE;
       "Avarii".avarie_motor := FALSE;
       "Avarii".avarie_greutate := FALSE;
   END_IF;
   "timer_reset_avarie_generala".TON(IN := "Avarii".reset_avarie_generala, PT := T#1s);
   IF "timer_reset_avarie_generala".Q THEN "Avarii".reset_avarie_generala := FALSE; END_IF;
END_REGION

REGION Network 6: Bec
   RUNG wire#powerrail
      "Bec_DB_1"(permisiune_pornire := "Bec_DB".permisiune_pornire, bec_aprins => "Bec_DB".led_aprins)
   END_RUNG
   // the same network as SCL:
   "Bec_DB_1"(permisiune_pornire := "Bec_DB".permisiune_pornire, bec_aprins => "Bec_DB".led_aprins);   // "Bec"
END_REGION

REGION Network 7: Usi
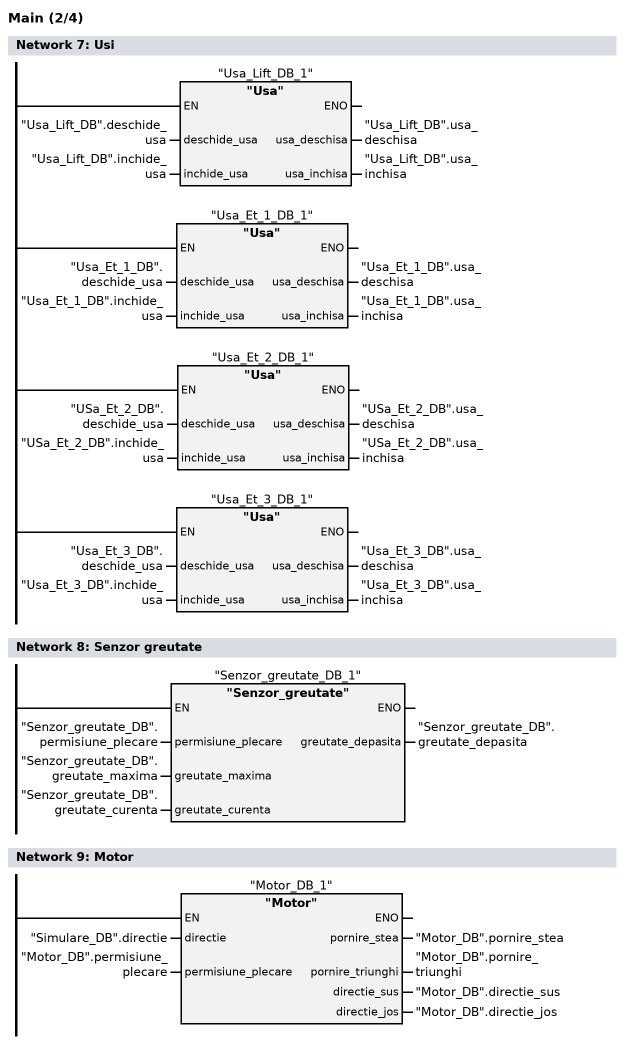
   RUNG wire#powerrail
      "Usa_Lift_DB_1"(deschide_usa := "Usa_Lift_DB".deschide_usa, inchide_usa := "Usa_Lift_DB".inchide_usa, usa_deschisa => "Usa_Lift_DB".usa_deschisa, usa_inchisa => "Usa_Lift_DB".usa_inchisa)
   END_RUNG
   RUNG wire#powerrail
      "Usa_Et_1_DB_1"(deschide_usa := "Usa_Et_1_DB".deschide_usa, inchide_usa := "Usa_Et_1_DB".inchide_usa, usa_deschisa => "Usa_Et_1_DB".usa_deschisa, usa_inchisa => "Usa_Et_1_DB".usa_inchisa)
   END_RUNG
   RUNG wire#powerrail
      "Usa_Et_2_DB_1"(deschide_usa := "USa_Et_2_DB".deschide_usa, inchide_usa := "USa_Et_2_DB".inchide_usa, usa_deschisa => "USa_Et_2_DB".usa_deschisa, usa_inchisa => "USa_Et_2_DB".usa_inchisa)
   END_RUNG
   RUNG wire#powerrail
      "Usa_Et_3_DB_1"(deschide_usa := "Usa_Et_3_DB".deschide_usa, inchide_usa := "Usa_Et_3_DB".inchide_usa, usa_deschisa => "Usa_Et_3_DB".usa_deschisa, usa_inchisa => "Usa_Et_3_DB".usa_inchisa)
   END_RUNG
   // the same network as SCL:
   "Usa_Lift_DB_1"(deschide_usa := "Usa_Lift_DB".deschide_usa,   // "Usa"
                   inchide_usa := "Usa_Lift_DB".inchide_usa,
                   usa_deschisa => "Usa_Lift_DB".usa_deschisa,
                   usa_inchisa => "Usa_Lift_DB".usa_inchisa);
   "Usa_Et_1_DB_1"(deschide_usa := "Usa_Et_1_DB".deschide_usa,   // "Usa"
                   inchide_usa := "Usa_Et_1_DB".inchide_usa,
                   usa_deschisa => "Usa_Et_1_DB".usa_deschisa,
                   usa_inchisa => "Usa_Et_1_DB".usa_inchisa);
   "Usa_Et_2_DB_1"(deschide_usa := "USa_Et_2_DB".deschide_usa,   // "Usa"
                   inchide_usa := "USa_Et_2_DB".inchide_usa,
                   usa_deschisa => "USa_Et_2_DB".usa_deschisa,
                   usa_inchisa => "USa_Et_2_DB".usa_inchisa);
   "Usa_Et_3_DB_1"(deschide_usa := "Usa_Et_3_DB".deschide_usa,   // "Usa"
                   inchide_usa := "Usa_Et_3_DB".inchide_usa,
                   usa_deschisa => "Usa_Et_3_DB".usa_deschisa,
                   usa_inchisa => "Usa_Et_3_DB".usa_inchisa);
END_REGION

REGION Network 8: Senzor greutate
   RUNG wire#powerrail
      "Senzor_greutate_DB_1"(permisiune_plecare := "Senzor_greutate_DB".permisiune_plecare, greutate_maxima := "Senzor_greutate_DB".greutate_maxima, greutate_curenta := "Senzor_greutate_DB".greutate_curenta, greutate_depasita => "Senzor_greutate_DB".greutate_depasita)
   END_RUNG
   // the same network as SCL:
   "Senzor_greutate_DB_1"(permisiune_plecare := "Senzor_greutate_DB".permisiune_plecare,   // "Senzor_greutate"
                          greutate_maxima := "Senzor_greutate_DB".greutate_maxima,
                          greutate_curenta := "Senzor_greutate_DB".greutate_curenta,
                          greutate_depasita => "Senzor_greutate_DB".greutate_depasita);
END_REGION

REGION Network 9: Motor
   RUNG wire#powerrail
      "Motor_DB_1"(directie := "Simulare_DB".directie, permisiune_plecare := "Motor_DB".permisiune_plecare, pornire_stea => "Motor_DB".pornire_stea, pornire_triunghi => "Motor_DB".pornire_triunghi, directie_sus => "Motor_DB".directie_sus, directie_jos => "Motor_DB".directie_jos)
   END_RUNG
   // the same network as SCL:
   "Motor_DB_1"(directie := "Simulare_DB".directie,   // "Motor"
                permisiune_plecare := "Motor_DB".permisiune_plecare,
                pornire_stea => "Motor_DB".pornire_stea,
                pornire_triunghi => "Motor_DB".pornire_triunghi,
                directie_sus => "Motor_DB".directie_sus,
                directie_jos => "Motor_DB".directie_jos);
END_REGION

REGION Network 10: Simulare
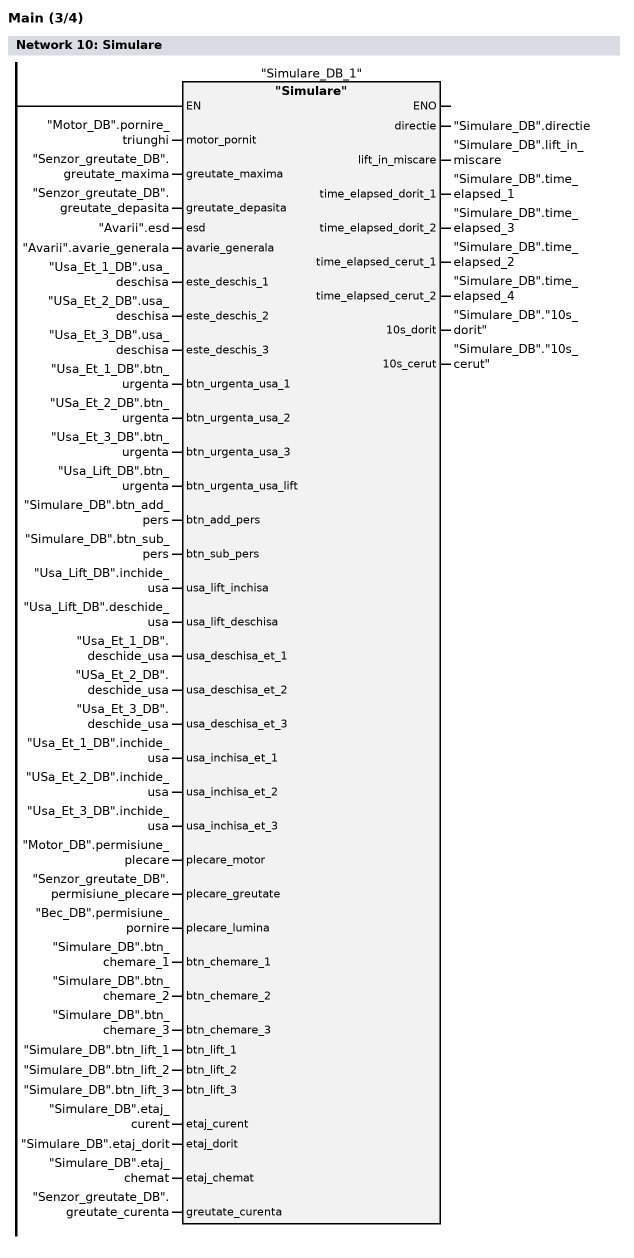
   RUNG wire#powerrail
      "Simulare_DB_1"(motor_pornit := "Motor_DB".pornire_triunghi, greutate_maxima := "Senzor_greutate_DB".greutate_maxima, greutate_depasita := "Senzor_greutate_DB".greutate_depasita, esd := "Avarii".esd, avarie_generala := "Avarii".avarie_generala, este_deschis_1 := "Usa_Et_1_DB".usa_deschisa, este_deschis_2 := "USa_Et_2_DB".usa_deschisa, este_deschis_3 := "Usa_Et_3_DB".usa_deschisa, btn_urgenta_usa_1 := "Usa_Et_1_DB".btn_urgenta, btn_urgenta_usa_2 := "USa_Et_2_DB".btn_urgenta, btn_urgenta_usa_3 := "Usa_Et_3_DB".btn_urgenta, btn_urgenta_usa_lift := "Usa_Lift_DB".btn_urgenta, btn_add_pers := "Simulare_DB".btn_add_pers, btn_sub_pers := "Simulare_DB".btn_sub_pers, usa_lift_inchisa := "Usa_Lift_DB".inchide_usa, usa_lift_deschisa := "Usa_Lift_DB".deschide_usa, usa_deschisa_et_1 := "Usa_Et_1_DB".deschide_usa, usa_deschisa_et_2 := "USa_Et_2_DB".deschide_usa, usa_deschisa_et_3 := "Usa_Et_3_DB".deschide_usa, usa_inchisa_et_1 := "Usa_Et_1_DB".inchide_usa, usa_inchisa_et_2 := "USa_Et_2_DB".inchide_usa, usa_inchisa_et_3 := "Usa_Et_3_DB".inchide_usa, plecare_motor := "Motor_DB".permisiune_plecare, plecare_greutate := "Senzor_greutate_DB".permisiune_plecare, plecare_lumina := "Bec_DB".permisiune_pornire, btn_chemare_1 := "Simulare_DB".btn_chemare_1, btn_chemare_2 := "Simulare_DB".btn_chemare_2, btn_chemare_3 := "Simulare_DB".btn_chemare_3, btn_lift_1 := "Simulare_DB".btn_lift_1, btn_lift_2 := "Simulare_DB".btn_lift_2, btn_lift_3 := "Simulare_DB".btn_lift_3, etaj_curent := "Simulare_DB".etaj_curent, etaj_dorit := "Simulare_DB".etaj_dorit, etaj_chemat := "Simulare_DB".etaj_chemat, greutate_curenta := "Senzor_greutate_DB".greutate_curenta, directie => "Simulare_DB".directie, lift_in_miscare => "Simulare_DB".lift_in_miscare, time_elapsed_dorit_1 => "Simulare_DB".time_elapsed_1, time_elapsed_dorit_2 => "Simulare_DB".time_elapsed_3, time_elapsed_cerut_1 => "Simulare_DB".time_elapsed_2, time_elapsed_cerut_2 => "Simulare_DB".time_elapsed_4, "10s_dorit" => "Simulare_DB"."10s_dorit", "10s_cerut" => "Simulare_DB"."10s_cerut")
   END_RUNG
   // the same network as SCL:
   "Simulare_DB_1"(motor_pornit := "Motor_DB".pornire_triunghi,   // "Simulare"
                   greutate_maxima := "Senzor_greutate_DB".greutate_maxima,
                   greutate_depasita := "Senzor_greutate_DB".greutate_depasita,
                   esd := "Avarii".esd,
                   avarie_generala := "Avarii".avarie_generala,
                   este_deschis_1 := "Usa_Et_1_DB".usa_deschisa,
                   este_deschis_2 := "USa_Et_2_DB".usa_deschisa,
                   este_deschis_3 := "Usa_Et_3_DB".usa_deschisa,
                   btn_urgenta_usa_1 := "Usa_Et_1_DB".btn_urgenta,
                   btn_urgenta_usa_2 := "USa_Et_2_DB".btn_urgenta,
                   btn_urgenta_usa_3 := "Usa_Et_3_DB".btn_urgenta,
                   btn_urgenta_usa_lift := "Usa_Lift_DB".btn_urgenta,
                   btn_add_pers := "Simulare_DB".btn_add_pers,
                   btn_sub_pers := "Simulare_DB".btn_sub_pers,
                   usa_lift_inchisa := "Usa_Lift_DB".inchide_usa,
                   usa_lift_deschisa := "Usa_Lift_DB".deschide_usa,
                   usa_deschisa_et_1 := "Usa_Et_1_DB".deschide_usa,
                   usa_deschisa_et_2 := "USa_Et_2_DB".deschide_usa,
                   usa_deschisa_et_3 := "Usa_Et_3_DB".deschide_usa,
                   usa_inchisa_et_1 := "Usa_Et_1_DB".inchide_usa,
                   usa_inchisa_et_2 := "USa_Et_2_DB".inchide_usa,
                   usa_inchisa_et_3 := "Usa_Et_3_DB".inchide_usa,
                   plecare_motor := "Motor_DB".permisiune_plecare,
                   plecare_greutate := "Senzor_greutate_DB".permisiune_plecare,
                   plecare_lumina := "Bec_DB".permisiune_pornire,
                   btn_chemare_1 := "Simulare_DB".btn_chemare_1,
                   btn_chemare_2 := "Simulare_DB".btn_chemare_2,
                   btn_chemare_3 := "Simulare_DB".btn_chemare_3,
                   btn_lift_1 := "Simulare_DB".btn_lift_1,
                   btn_lift_2 := "Simulare_DB".btn_lift_2,
                   btn_lift_3 := "Simulare_DB".btn_lift_3,
                   etaj_curent := "Simulare_DB".etaj_curent,
                   etaj_dorit := "Simulare_DB".etaj_dorit,
                   etaj_chemat := "Simulare_DB".etaj_chemat,
                   greutate_curenta := "Senzor_greutate_DB".greutate_curenta,
                   directie => "Simulare_DB".directie,
                   lift_in_miscare => "Simulare_DB".lift_in_miscare,
                   time_elapsed_dorit_1 => "Simulare_DB".time_elapsed_1,
                   time_elapsed_dorit_2 => "Simulare_DB".time_elapsed_3,
                   time_elapsed_cerut_1 => "Simulare_DB".time_elapsed_2,
                   time_elapsed_cerut_2 => "Simulare_DB".time_elapsed_4,
                   "10s_dorit" => "Simulare_DB"."10s_dorit",
                   "10s_cerut" => "Simulare_DB"."10s_cerut");
END_REGION

REGION Network 11: timer in secunde
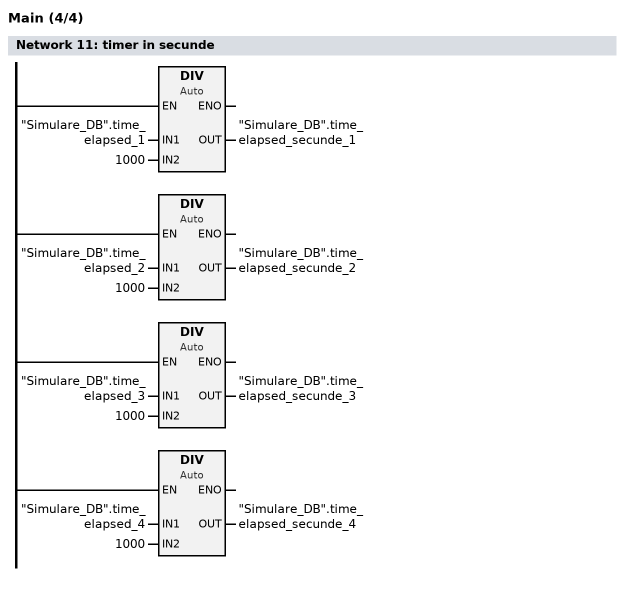
   RUNG wire#powerrail
      Div(in1 := "Simulare_DB".time_elapsed_1, in2 := 1000, out => "Simulare_DB".time_elapsed_secunde_1)
   END_RUNG
   RUNG wire#powerrail
      Div(in1 := "Simulare_DB".time_elapsed_2, in2 := 1000, out => "Simulare_DB".time_elapsed_secunde_2)
   END_RUNG
   RUNG wire#powerrail
      Div(in1 := "Simulare_DB".time_elapsed_3, in2 := 1000, out => "Simulare_DB".time_elapsed_secunde_3)
   END_RUNG
   RUNG wire#powerrail
      Div(in1 := "Simulare_DB".time_elapsed_4, in2 := 1000, out => "Simulare_DB".time_elapsed_secunde_4)
   END_RUNG
   // the same network as SCL:
   "Simulare_DB".time_elapsed_secunde_1 := "Simulare_DB".time_elapsed_1 / 1000;
   "Simulare_DB".time_elapsed_secunde_2 := "Simulare_DB".time_elapsed_2 / 1000;
   "Simulare_DB".time_elapsed_secunde_3 := "Simulare_DB".time_elapsed_3 / 1000;
   "Simulare_DB".time_elapsed_secunde_4 := "Simulare_DB".time_elapsed_4 / 1000;
END_REGION
END_ORGANIZATION_BLOCK

(* ===== HMI "HMI_RT_1" =====
system functions are stored by id; their names below are inferred from use
connection "HMI_Connection_1": ETHERNET, SMART_S7_1500_OMS

HMI tags "Default tag table"
   "Alarme_alarme_gather" : Word = PLC Alarme.alarme_gather, 1 s
   "Avarii_esd" : Bool = PLC Avarii.esd, 1 s
   "Avarii_btn_esd" : Bool = PLC Avarii.btn_esd, 1 s
   "Avarii_reset_esd" : Bool = PLC Avarii.reset_esd, 1 s
   "Avarii_avarie_usa" : Bool = PLC Avarii.avarie_usa, 1 s
   "Avarii_avarie_lumina" : Bool = PLC Avarii.avarie_lumina, 1 s
   "Avarii_avarie_motor" : Bool = PLC Avarii.avarie_motor, 1 s
   "Avarii_avarie_greutate" : Bool = PLC Avarii.avarie_greutate, 1 s
   "Avarii_reset_avarie_generala" : Bool = PLC Avarii.reset_avarie_generala, 1 s
   "Simulare_DB_btn_chemare_3" : Bool = PLC Simulare_DB.btn_chemare_3, 1 s
   "Simulare_DB_btn_chemare_2" : Bool = PLC Simulare_DB.btn_chemare_2, 1 s
   "Simulare_DB_btn_chemare_1" : Bool = PLC Simulare_DB.btn_chemare_1, 1 s
   "Simulare_DB_lift_in_miscare" : Bool = PLC Simulare_DB.lift_in_miscare, 1 s
   "Senzor_greutate_DB_greutate_depasita" : Bool = PLC Senzor_greutate_DB.greutate_depasita, 1 s
   "Simulare_DB_btn_add_pers" : Bool = PLC Simulare_DB.btn_add_pers, 1 s
   "Simulare_DB_btn_sub_pers" : Bool = PLC Simulare_DB.btn_sub_pers, 1 s
   "Senzor_greutate_DB_greutate_curenta" : Real = PLC Senzor_greutate_DB.greutate_curenta, 1 s
   "Motor_DB_directie_sus" : Bool = PLC Motor_DB.directie_sus, 1 s
   "Motor_DB_directie_jos" : Bool = PLC Motor_DB.directie_jos, 1 s
   "Simulare_DB_btn_lift_2" : Bool = PLC Simulare_DB.btn_lift_2, 1 s
   "Simulare_DB_btn_lift_3" : Bool = PLC Simulare_DB.btn_lift_3, 1 s
   "Simulare_DB_btn_lift_1" : Bool = PLC Simulare_DB.btn_lift_1, 1 s
   "Simulare_DB_etaj_curent" : Int = PLC Simulare_DB.etaj_curent, 1 s
   "Bec_DB_led_aprins" : Bool = PLC Bec_DB.led_aprins, 1 s
   "Senzor_greutate_DB_permisiune_plecare" : Bool = PLC Senzor_greutate_DB.permisiune_plecare, 1 s
   "Motor_DB_pornire_stea" : Bool = PLC Motor_DB.pornire_stea, 1 s
   "Motor_DB_pornire_triunghi" : Bool = PLC Motor_DB.pornire_triunghi, 1 s
   "Usa_Lift_DB_deschide_usa" : Bool = PLC Usa_Lift_DB.deschide_usa, 1 s
   "Usa_Lift_DB_usa_deschisa" : Bool = PLC Usa_Lift_DB.usa_deschisa, 1 s
   "Usa_Lift_DB_usa_inchisa" : Bool = PLC Usa_Lift_DB.usa_inchisa, 1 s
   "Usa_Et_1_DB_usa_deschisa" : Bool = PLC Usa_Et_1_DB.usa_deschisa, 1 s
   "USa_Et_2_DB_usa_deschisa" : Bool = PLC USa_Et_2_DB.usa_deschisa, 1 s
   "Usa_Et_3_DB_usa_deschisa" : Bool = PLC Usa_Et_3_DB.usa_deschisa, 1 s
   "Usa_Lift_DB_btn_urgenta" : Bool = PLC Usa_Lift_DB.btn_urgenta, 1 s
   "Usa_Et_1_DB_btn_urgenta" : Bool = PLC Usa_Et_1_DB.btn_urgenta, 1 s
   "Usa_Et_3_DB_btn_urgenta" : Bool = PLC Usa_Et_3_DB.btn_urgenta, 1 s
   "USa_Et_2_DB_btn_urgenta" : Bool = PLC USa_Et_2_DB.btn_urgenta, 1 s
   "Simulare_DB_time_elapsed_secunde_1" : Time = PLC Simulare_DB.time_elapsed_secunde_1, 1 s
   "Simulare_DB_time_elapsed_secunde_2" : Time = PLC Simulare_DB.time_elapsed_secunde_2, 1 s
   "Simulare_DB_time_elapsed_secunde_3" : Time = PLC Simulare_DB.time_elapsed_secunde_3, 1 s
   "Simulare_DB_time_elapsed_secunde_4" : Time = PLC Simulare_DB.time_elapsed_secunde_4, 1 s
   "Simulare_DB_10s_cerut" : Bool = PLC Simulare_DB.10s_cerut, 1 s
   "Simulare_DB_10s_dorit" : Bool = PLC Simulare_DB.10s_dorit, 1 s

discrete alarms
   1: 'ESD', class Errors, trigger "Alarme_alarme_gather" bit 0
   2: 'Avarie la usa', class Errors, trigger "Alarme_alarme_gather" bit 1
   3: 'Avarie la bec', class Errors, trigger "Alarme_alarme_gather" bit 2
   4: 'Avarie la motor', class Errors, trigger "Alarme_alarme_gather" bit 3
   5: 'Avarie la senzorul de greutate', class Errors, trigger "Alarme_alarme_gather" bit 4
   6: 'Greutate maxiam atinsa/depasita', class Errors, trigger "Alarme_alarme_gather" bit 5

Template "Template_1" 800x480
   Button "Exit" at 722,440 size 55x39; TextOff 'Exit'; PictureOff "ExitRuntime_KTP900_Basic_PN_TR"; PictureOn "ExitRuntime_KTP900_Basic_PN_TR"
      on Release: StopRuntime(0)

screen "Et1" 800x480, template "Template_1"
   Rectangle "Rectangle_12" at 353,101 size 186x286
      Visibility <- "Usa_Lift_DB_usa_inchisa"
   TextField "Text field_1" at 34,456 size 42x20; Text 'Etaj 1'
   TextField "Text field_2" at 130,457 size 42x20; Text 'Etaj 2'
   TextField "Text field_3" at 226,457 size 42x20; Text 'Etaj 3'
   TextField "Text field_4" at 325,457 size 51x20; Text 'Alarme'
   Button "Button_1" at 47,35 size 49x27; TextOff 'ESD'
      on Click: SetBit("Avarii_btn_esd")
   Button "Button_2" at 107,35 size 49x27; TextOff 'Reset'
      on Click: SetBit("Avarii_reset_esd")
   Circle "Circle_1" at 7,35 size 28x28
      Appearance <- "Avarii_esd"
   Button "Button_3" at 47,81 size 49x27; TextOff 'Usa'
      on Click: SetBit("Avarii_avarie_usa")
   Button "Button_4" at 47,128 size 49x27; TextOff 'Bec'
      on Click: SetBit("Avarii_avarie_lumina")
   Button "Button_5" at 47,175 size 49x27; TextOff 'Motor'
      on Click: SetBit("Avarii_avarie_motor")
   Button "Button_6" at 47,222 size 49x27; TextOff 'Greu.'
      on Click: SetBit("Avarii_avarie_greutate")
   Button "Button_7" at 107,155 size 49x27; TextOff 'Reset'
      on Click: SetBit("Avarii_reset_avarie_generala")
   Circle "Circle_2" at 7,78 size 28x28
      Appearance <- "Avarii_avarie_usa"
   Circle "Circle_3" at 7,126 size 28x28
      Appearance <- "Avarii_avarie_lumina"
   Circle "Circle_4" at 7,172 size 28x28
      Appearance <- "Avarii_avarie_motor"
   Circle "Circle_5" at 7,219 size 28x28
      Appearance <- "Avarii_avarie_greutate"
   Rectangle "Rectangle_2" at 353,101 size 186x286
      Visibility <- "Usa_Lift_DB_usa_deschisa"
   TextField "Text field_5" at 365,19 size 67x29; Text 'Etaj 1'
   TextField "Text field_6" at 413,181 size 65x20; Text 'Lift (Usa)'
   TextField "Text field_7" at 239,182 size 58x20; Text 'Usa etaj'
   Rectangle "Rectangle_4" at 538,238 size 37x75
      Visibility <- "Motor_DB_pornire_stea"
      Appearance <- "Motor_DB_pornire_stea"
   TextField "Text field_8" at 575,261 size 44x20; Text 'Motor'
   Circle "Circle_6" at 426,101 size 33x33
      Appearance <- "Bec_DB_led_aprins"
   TextField "Text field_9" at 428,129 size 28x20; Text 'Bec'
   TextField "Text field_10" at 390,410 size 112x20; Text 'Senzor greutate'
   IOField "I/O field_1" at 713,48 size 72x32; FormatPattern 99
      ProcessValue <- "Simulare_DB_etaj_curent"
   TextField "Text field_11" at 708,28 size 77x20; Text 'Etaj curent'
   IOField "I/O field_2" at 713,106 size 74x32; FormatPattern 99; Unit s
      ProcessValue <- "Simulare_DB_time_elapsed_secunde_2"
   TextField "Text field_12" at 708,86 size 79x20; Text 'Timp venire'
   IOField "I/O field_3" at 713,222 size 75x32; FormatPattern 999.99; Unit kg
      ProcessValue <- "Senzor_greutate_DB_greutate_curenta"
   TextField "Text field_13" at 708,202 size 63x20; Text 'Greutate'
   Button "Button_8" at 456,438 size 42x32; TextOff 'Add'
      on Click: SetBit("Simulare_DB_btn_add_pers")
   Button "Button_9" at 513,438 size 42x32; TextOff 'Sub'
      on Click: SetBit("Simulare_DB_btn_sub_pers")
   Button "Button_10" at 353,275 size 36x32; TextOff 'Et 2'
      on Click: SetBit("Simulare_DB_btn_lift_2")
   Button "Button_11" at 353,314 size 36x32; TextOff 'Et 3'
      on Click: SetBit("Simulare_DB_btn_lift_3")
   Button "Button_12" at 82,344 size 96x32; TextOff 'Cheama'
      on Click: SetBit("Simulare_DB_btn_chemare_1")
   Rectangle "Rectangle_6" at 538,112 size 39x22
      Appearance <- "Motor_DB_directie_sus"
   TextField "Text field_14" at 541,112 size 28x20; Text 'Sus'
   Rectangle "Rectangle_7" at 538,133 size 39x22
      Appearance <- "Motor_DB_directie_jos"
   TextField "Text field_15" at 542,133 size 26x20; Text 'Jos'
   Rectangle "Rectangle_8" at 370,82 size 146x20
      Appearance <- "Simulare_DB_lift_in_miscare"
   TextField "Text field_16" at 397,64 size 95x20; Text 'Lift in miscare'
   Circle "Circle_7" at 713,285 size 39x39
      Visibility <- "Senzor_greutate_DB_greutate_depasita"
   TextField "Text field_17" at 671,265 size 123x20; Text 'Greutate depasita'
      Visibility <- "Senzor_greutate_DB_greutate_depasita"
   Rectangle "Rectangle_5" at 372,386 size 146x27
      Appearance <- "Senzor_greutate_DB_permisiune_plecare"
   Rectangle "Rectangle_9" at 538,238 size 37x75
      Appearance <- "Motor_DB_pornire_triunghi"
      Visibility <- "Motor_DB_pornire_triunghi"
   Rectangle "Rectangle_11" at 310,102 size 33x285
      Visibility <- "Usa_Et_1_DB_usa_deschisa"
   Button "Button_13" at 503,275 size 36x32; TextOff 'Usa'
      on Click: SetBit("Usa_Lift_DB_btn_urgenta")
      Visibility <- "Avarii_esd"
   Button "Button_17" at 245,207 size 46x32; TextOff 'Usa'
      on Click: SetBit("Usa_Et_1_DB_btn_urgenta")
      Visibility <- "Avarii_esd"
   IOField "I/O field_4" at 713,163 size 74x32; FormatPattern 99; Unit s
      ProcessValue <- "Simulare_DB_time_elapsed_secunde_1"
   TextField "Text field_18" at 708,143 size 73x20; Text 'Timp ajuns'
   IOField "I/O field_5" at 713,163 size 73x32; FormatPattern 99; Unit s
      ProcessValue <- "Simulare_DB_time_elapsed_secunde_3"
      Visibility <- "Simulare_DB_10s_dorit"
   IOField "I/O field_6" at 714,107 size 73x32; FormatPattern 99; Unit s
      ProcessValue <- "Simulare_DB_time_elapsed_secunde_4"
      Visibility <- "Simulare_DB_10s_cerut"

screen "Et2" 800x480
   Rectangle "Rectangle_12" at 353,101 size 186x286
      Visibility <- "Usa_Lift_DB_usa_inchisa"
   Rectangle "Rectangle_2" at 353,101 size 186x286
      Visibility <- "Usa_Lift_DB_usa_deschisa"
   TextField "Text field_1" at 34,456 size 42x20; Text 'Etaj 1'
   TextField "Text field_2" at 130,457 size 42x20; Text 'Etaj 2'
   TextField "Text field_3" at 226,457 size 42x20; Text 'Etaj 3'
   TextField "Text field_4" at 325,457 size 51x20; Text 'Alarme'
   TextField "Text field_5" at 365,19 size 67x29; Text 'Etaj 2'
   TextField "Text field_11" at 708,28 size 77x20; Text 'Etaj curent'
   Button "Button_12" at 82,344 size 96x32; TextOff 'Cheama'
      on Click: SetBit("Simulare_DB_btn_chemare_2")
   TextField "Text field_6" at 413,181 size 65x20; Text 'Lift (Usa)'
   TextField "Text field_7" at 239,182 size 58x20; Text 'Usa etaj'
   TextField "Text field_8" at 575,261 size 44x20; Text 'Motor'
   TextField "Text field_9" at 428,129 size 28x20; Text 'Bec'
   TextField "Text field_10" at 390,410 size 112x20; Text 'Senzor greutate'
   Button "Button_10" at 353,275 size 36x32; TextOff 'Et 1'
      on Click: SetBit("Simulare_DB_btn_lift_1")
   Button "Button_11" at 353,314 size 36x32; TextOff 'Et 3'
      on Click: SetBit("Simulare_DB_btn_lift_3")
   Button "Button_1" at 47,35 size 49x27; TextOff 'ESD'
      on Click: SetBit("Avarii_btn_esd")
   Button "Button_2" at 107,35 size 49x27; TextOff 'Reset'
      on Click: SetBit("Avarii_reset_esd")
   Circle "Circle_1" at 7,35 size 28x28
      Appearance <- "Avarii_esd"
   Button "Button_3" at 47,81 size 49x27; TextOff 'Usa'
      on Click: SetBit("Avarii_avarie_usa")
   Button "Button_4" at 47,128 size 49x27; TextOff 'Bec'
      on Click: SetBit("Avarii_avarie_lumina")
   Button "Button_5" at 47,175 size 49x27; TextOff 'Motor'
      on Click: SetBit("Avarii_avarie_motor")
   Button "Button_6" at 47,222 size 49x27; TextOff 'Greu.'
      on Click: SetBit("Avarii_avarie_greutate")
   Button "Button_7" at 107,155 size 49x27; TextOff 'Reset'
      on Click: SetBit("Avarii_reset_avarie_generala")
   Circle "Circle_2" at 7,78 size 28x28
      Appearance <- "Avarii_avarie_usa"
   Circle "Circle_3" at 7,126 size 28x28
      Appearance <- "Avarii_avarie_lumina"
   Circle "Circle_4" at 7,172 size 28x28
      Appearance <- "Avarii_avarie_motor"
   Circle "Circle_5" at 7,219 size 28x28
      Appearance <- "Avarii_avarie_greutate"
   Rectangle "Rectangle_8" at 370,82 size 146x20
      Appearance <- "Simulare_DB_lift_in_miscare"
   TextField "Text field_16" at 397,64 size 95x20; Text 'Lift in miscare'
   Button "Button_8" at 456,438 size 42x32; TextOff 'Add'
      on Click: SetBit("Simulare_DB_btn_add_pers")
   Button "Button_9" at 513,438 size 42x32; TextOff 'Sub'
      on Click: SetBit("Simulare_DB_btn_sub_pers")
   Rectangle "Rectangle_6" at 538,112 size 39x22
      Appearance <- "Motor_DB_directie_sus"
   TextField "Text field_14" at 541,112 size 28x20; Text 'Sus'
   Rectangle "Rectangle_7" at 538,133 size 39x22
      Appearance <- "Motor_DB_directie_jos"
   TextField "Text field_15" at 542,133 size 26x20; Text 'Jos'
   IOField "I/O field_1" at 713,48 size 72x32; FormatPattern 99
      ProcessValue <- "Simulare_DB_etaj_curent"
   Circle "Circle_6" at 426,101 size 33x33
      Appearance <- "Bec_DB_led_aprins"
   Rectangle "Rectangle_5" at 372,386 size 146x27
      Appearance <- "Senzor_greutate_DB_permisiune_plecare"
   Rectangle "Rectangle_9" at 538,238 size 37x75
      Visibility <- "Motor_DB_pornire_stea"
      Appearance <- "Motor_DB_pornire_stea"
   Rectangle "Rectangle_10" at 538,238 size 37x75
      Visibility <- "Motor_DB_pornire_triunghi"
      Appearance <- "Motor_DB_pornire_triunghi"
   Rectangle "Rectangle_11" at 310,102 size 33x285
      Visibility <- "USa_Et_2_DB_usa_deschisa"
   Button "Button_13" at 503,275 size 36x32; TextOff 'Usa'
      on Click: SetBit("Usa_Lift_DB_btn_urgenta")
      Visibility <- "Avarii_esd"
   Button "Button_17" at 245,207 size 46x32; TextOff 'Usa'
      on Click: SetBit("USa_Et_2_DB_btn_urgenta")
      Visibility <- "Avarii_esd"
   IOField "I/O field_2" at 713,106 size 74x32; FormatPattern 99; Unit s
      ProcessValue <- "Simulare_DB_time_elapsed_secunde_2"
   TextField "Text field_12" at 708,86 size 79x20; Text 'Timp venire'
   IOField "I/O field_3" at 713,222 size 75x32; FormatPattern 999.99; Unit kg
      ProcessValue <- "Senzor_greutate_DB_greutate_curenta"
   TextField "Text field_13" at 708,202 size 63x20; Text 'Greutate'
   Circle "Circle_7" at 713,285 size 39x39
      Visibility <- "Senzor_greutate_DB_greutate_depasita"
   TextField "Text field_17" at 671,265 size 123x20; Text 'Greutate depasita'
      Visibility <- "Senzor_greutate_DB_greutate_depasita"
   IOField "I/O field_4" at 713,163 size 74x32; FormatPattern 99; Unit s
      ProcessValue <- "Simulare_DB_time_elapsed_secunde_1"
   TextField "Text field_18" at 708,143 size 73x20; Text 'Timp ajuns'
   IOField "I/O field_5" at 714,163 size 73x32; FormatPattern 99; Unit s
      Visibility <- "Simulare_DB_10s_dorit"
      ProcessValue <- "Simulare_DB_time_elapsed_secunde_3"
   IOField "I/O field_6" at 713,107 size 73x32; FormatPattern 99; Unit s
      Visibility <- "Simulare_DB_10s_cerut"
      ProcessValue <- "Simulare_DB_time_elapsed_secunde_4"

screen "Et3" 800x480
   Rectangle "Rectangle_12" at 353,101 size 186x286
      Visibility <- "Usa_Lift_DB_usa_inchisa"
   Rectangle "Rectangle_2" at 353,101 size 186x286
      Visibility <- "Usa_Lift_DB_usa_deschisa"
   TextField "Text field_1" at 34,456 size 42x20; Text 'Etaj 1'
   TextField "Text field_2" at 130,457 size 42x20; Text 'Etaj 2'
   TextField "Text field_3" at 226,457 size 42x20; Text 'Etaj 3'
   TextField "Text field_4" at 325,457 size 51x20; Text 'Alarme'
   TextField "Text field_5" at 365,19 size 67x29; Text 'Etaj 3'
   TextField "Text field_11" at 708,28 size 77x20; Text 'Etaj curent'
   Button "Button_12" at 82,344 size 96x32; TextOff 'Cheama'
      on Click: SetBit("Simulare_DB_btn_chemare_3")
   TextField "Text field_6" at 413,181 size 65x20; Text 'Lift (Usa)'
   TextField "Text field_7" at 239,182 size 58x20; Text 'Usa etaj'
   TextField "Text field_8" at 575,261 size 44x20; Text 'Motor'
   TextField "Text field_9" at 428,129 size 28x20; Text 'Bec'
   Rectangle "Rectangle_5" at 372,386 size 146x27
      Appearance <- "Senzor_greutate_DB_permisiune_plecare"
   TextField "Text field_10" at 390,410 size 112x20; Text 'Senzor greutate'
   Button "Button_10" at 353,275 size 36x32; TextOff 'Et 1'
      on Click: SetBit("Simulare_DB_btn_lift_1")
   Button "Button_11" at 353,314 size 36x32; TextOff 'Et 2'
      on Click: SetBit("Simulare_DB_btn_lift_2")
   Button "Button_13" at 503,275 size 36x32; TextOff 'Usa'
      Visibility <- "Avarii_esd"
      on Click: SetBit("Usa_Lift_DB_btn_urgenta")
   Button "Button_17" at 245,207 size 46x32; TextOff 'Usa'
      Visibility <- "Avarii_esd"
      on Click: SetBit("Usa_Et_3_DB_btn_urgenta")
   Button "Button_1" at 47,35 size 49x27; TextOff 'ESD'
      on Click: SetBit("Avarii_btn_esd")
   Button "Button_2" at 107,35 size 49x27; TextOff 'Reset'
      on Click: SetBit("Avarii_reset_esd")
   Circle "Circle_1" at 7,35 size 28x28
      Appearance <- "Avarii_esd"
   Button "Button_3" at 47,81 size 49x27; TextOff 'Usa'
      on Click: SetBit("Avarii_avarie_usa")
   Button "Button_4" at 47,128 size 49x27; TextOff 'Bec'
      on Click: SetBit("Avarii_avarie_lumina")
   Button "Button_5" at 47,175 size 49x27; TextOff 'Motor'
      on Click: SetBit("Avarii_avarie_motor")
   Button "Button_6" at 47,222 size 49x27; TextOff 'Greu.'
      on Click: SetBit("Avarii_avarie_greutate")
   Button "Button_7" at 107,155 size 49x27; TextOff 'Reset'
      on Click: SetBit("Avarii_reset_avarie_generala")
   Circle "Circle_2" at 7,78 size 28x28
      Appearance <- "Avarii_avarie_usa"
   Circle "Circle_3" at 7,126 size 28x28
      Appearance <- "Avarii_avarie_lumina"
   Circle "Circle_4" at 7,172 size 28x28
      Appearance <- "Avarii_avarie_motor"
   Circle "Circle_5" at 7,219 size 28x28
      Appearance <- "Avarii_avarie_greutate"
   Rectangle "Rectangle_8" at 370,82 size 146x20
      Appearance <- "Simulare_DB_lift_in_miscare"
   TextField "Text field_16" at 397,64 size 95x20; Text 'Lift in miscare'
   Button "Button_8" at 456,438 size 42x32; TextOff 'Add'
      on Click: SetBit("Simulare_DB_btn_add_pers")
   Button "Button_9" at 513,438 size 42x32; TextOff 'Sub'
      on Click: SetBit("Simulare_DB_btn_sub_pers")
   Rectangle "Rectangle_6" at 538,112 size 39x22
      Appearance <- "Motor_DB_directie_sus"
   TextField "Text field_14" at 541,112 size 28x20; Text 'Sus'
   Rectangle "Rectangle_7" at 538,133 size 39x22
      Appearance <- "Motor_DB_directie_jos"
   TextField "Text field_15" at 542,133 size 26x20; Text 'Jos'
   IOField "I/O field_1" at 713,48 size 72x32; FormatPattern 99
      ProcessValue <- "Simulare_DB_etaj_curent"
   Circle "Circle_6" at 426,101 size 33x33
      Appearance <- "Bec_DB_led_aprins"
   Rectangle "Rectangle_9" at 538,238 size 37x75
      Visibility <- "Motor_DB_pornire_stea"
      Appearance <- "Motor_DB_pornire_stea"
   Rectangle "Rectangle_10" at 538,238 size 37x75
      Visibility <- "Motor_DB_pornire_triunghi"
      Appearance <- "Motor_DB_pornire_triunghi"
   Rectangle "Rectangle_11" at 310,102 size 33x285
      Visibility <- "Usa_Et_3_DB_usa_deschisa"
   IOField "I/O field_2" at 713,106 size 74x32; FormatPattern 99; Unit s
      ProcessValue <- "Simulare_DB_time_elapsed_secunde_2"
   TextField "Text field_12" at 708,86 size 79x20; Text 'Timp venire'
   IOField "I/O field_3" at 713,222 size 75x32; FormatPattern 999.99; Unit kg
      ProcessValue <- "Senzor_greutate_DB_greutate_curenta"
   TextField "Text field_13" at 708,202 size 63x20; Text 'Greutate'
   Circle "Circle_7" at 713,285 size 39x39
      Visibility <- "Senzor_greutate_DB_greutate_depasita"
   TextField "Text field_17" at 671,265 size 123x20; Text 'Greutate depasita'
      Visibility <- "Senzor_greutate_DB_greutate_depasita"
   IOField "I/O field_4" at 713,163 size 74x32; FormatPattern 99; Unit s
      ProcessValue <- "Simulare_DB_time_elapsed_secunde_1"
   TextField "Text field_18" at 708,143 size 73x20; Text 'Timp ajuns'
   IOField "I/O field_5" at 713,163 size 73x32; FormatPattern 99; Unit s
      Visibility <- "Simulare_DB_10s_dorit"
      ProcessValue <- "Simulare_DB_time_elapsed_secunde_3"
   IOField "I/O field_6" at 714,107 size 73x32; FormatPattern 99; Unit s
      Visibility <- "Simulare_DB_10s_cerut"
      ProcessValue <- "Simulare_DB_time_elapsed_secunde_4"
*)